LIN {X 745.357, Y -369.718, Z 305.5, A 0, B 90, C -0, E1 0, E2 0, E3 0, E4 0} C_DIS
LIN {X 743.421, Y -368.973, Z 305.5, A 0, B 90, C -0, E1 0, E2 0, E3 0, E4 0} C_DIS
LIN {X 741.486, Y -368.227, Z 305.5, A 0, B 90, C -0, E1 0, E2 0, E3 0, E4 0} C_DIS
LIN {X 739.55, Y -367.481, Z 305.5, A 0, B 90, C -0, E1 0, E2 0, E3 0, E4 0} C_DIS
LIN {X 737.563, Y -367.409, Z 305.5, A 0, B 90, C -0, E1 0, E2 0, E3 0, E4 0} C_DIS
LIN {X 736.667, Y -369.222, Z 305.5, A 0, B 90, C -0, E1 0, E2 0, E3 0, E4 0} C_DIS
LIN {X 736.176, Y -371.238, Z 305.5, A 0, B 90, C -0, E1 0, E2 0, E3 0, E4 0} C_DIS
LIN {X 735.685, Y -373.253, Z 305.5, A 0, B 90, C -0, E1 0, E2 0, E3 0, E4 0} C_DIS
LIN {X 735.194, Y -375.268, Z 305.5, A 0, B 90, C -0, E1 0, E2 0, E3 0, E4 0} C_DIS
LIN {X 734.703, Y -377.283, Z 305.5, A 0, B 90, C -0, E1 0, E2 0, E3 0, E4 0} C_DIS
LIN {X 734.212, Y -379.299, Z 305.5, A 0, B 90, C -0, E1 0, E2 0, E3 0, E4 0} C_DIS
LIN {X 733.185, Y -381.059, Z 305.5, A 0, B 90, C -0, E1 0, E2 0, E3 0, E4 0} C_DIS
LIN {X 731.276, Y -381.793, Z 305.5, A 0, B 90, C -0, E1 0, E2 0, E3 0, E4 0} C_DIS
LIN {X 729.227, Y -382.115, Z 305.5, A 0, B 90, C -0, E1 0, E2 0, E3 0, E4 0} C_DIS
LIN {X 727.178, Y -382.437, Z 305.5, A 0, B 90, C -0, E1 0, E2 0, E3 0, E4 0} C_DIS
LIN {X 725.128, Y -382.759, Z 305.5, A 0, B 90, C -0, E1 0, E2 0, E3 0, E4 0} C_DIS
LIN {X 723.079, Y -383.081, Z 305.5, A 0, B 90, C -0, E1 0, E2 0, E3 0, E4 0} C_DIS
LIN {X 721.03, Y -383.402, Z 305.5, A 0, B 90, C -0, E1 0, E2 0, E3 0, E4 0} C_DIS
LIN {X 719.273, Y -384.334, Z 305.5, A 0, B 90, C -0, E1 0, E2 0, E3 0, E4 0} C_DIS
LIN {X 719.404, Y -386.352, Z 305.5, A 0, B 90, C -0, E1 0, E2 0, E3 0, E4 0} C_DIS
LIN {X 719.987, Y -388.343, Z 305.5, A 0, B 90, C -0, E1 0, E2 0, E3 0, E4 0} C_DIS
LIN {X 720.569, Y -390.334, Z 305.5, A 0, B 90, C -0, E1 0, E2 0, E3 0, E4 0} C_DIS
LIN {X 721.151, Y -392.324, Z 305.5, A 0, B 90, C -0, E1 0, E2 0, E3 0, E4 0} C_DIS
LIN {X 721.734, Y -394.315, Z 305.5, A 0, B 90, C -0, E1 0, E2 0, E3 0, E4 0} C_DIS
LIN {X 722.316, Y -396.306, Z 305.5, A 0, B 90, C -0, E1 0, E2 0, E3 0, E4 0} C_DIS
LIN {X 722.307, Y -398.344, Z 305.5, A 0, B 90, C -0, E1 0, E2 0, E3 0, E4 0} C_DIS
LIN {X 721.021, Y -399.934, Z 305.5, A 0, B 90, C -0, E1 0, E2 0, E3 0, E4 0} C_DIS
LIN {X 719.407, Y -401.237, Z 305.5, A 0, B 90, C -0, E1 0, E2 0, E3 0, E4 0} C_DIS
LIN {X 717.793, Y -402.541, Z 305.5, A 0, B 90, C -0, E1 0, E2 0, E3 0, E4 0} C_DIS
LIN {X 716.18, Y -403.844, Z 305.5, A 0, B 90, C -0, E1 0, E2 0, E3 0, E4 0} C_DIS
LIN {X 714.566, Y -405.147, Z 305.5, A 0, B 90, C -0, E1 0, E2 0, E3 0, E4 0} C_DIS
LIN {X 712.952, Y -406.451, Z 305.5, A 0, B 90, C -0, E1 0, E2 0, E3 0, E4 0} C_DIS
LIN {X 711.897, Y -408.136, Z 305.5, A 0, B 90, C -0, E1 0, E2 0, E3 0, E4 0} C_DIS
LIN {X 713.019, Y -409.818, Z 305.5, A 0, B 90, C -0, E1 0, E2 0, E3 0, E4 0} C_DIS
LIN {X 714.519, Y -411.251, Z 305.5, A 0, B 90, C -0, E1 0, E2 0, E3 0, E4 0} C_DIS
LIN {X 716.019, Y -412.684, Z 305.5, A 0, B 90, C -0, E1 0, E2 0, E3 0, E4 0} C_DIS
LIN {X 717.518, Y -414.117, Z 305.5, A 0, B 90, C -0, E1 0, E2 0, E3 0, E4 0} C_DIS
LIN {X 719.018, Y -415.55, Z 305.5, A 0, B 90, C -0, E1 0, E2 0, E3 0, E4 0} C_DIS
LIN {X 720.518, Y -416.982, Z 305.5, A 0, B 90, C -0, E1 0, E2 0, E3 0, E4 0} C_DIS
LIN {X 721.529, Y -418.752, Z 305.5, A 0, B 90, C -0, E1 0, E2 0, E3 0, E4 0} C_DIS
LIN {X 721.21, Y -420.772, Z 305.5, A 0, B 90, C -0, E1 0, E2 0, E3 0, E4 0} C_DIS
LIN {X 720.464, Y -422.708, Z 305.5, A 0, B 90, C -0, E1 0, E2 0, E3 0, E4 0} C_DIS
LIN {X 719.718, Y -424.643, Z 305.5, A 0, B 90, C -0, E1 0, E2 0, E3 0, E4 0} C_DIS
LIN {X 718.973, Y -426.579, Z 305.5, A 0, B 90, C -0, E1 0, E2 0, E3 0, E4 0} C_DIS
LIN {X 718.227, Y -428.514, Z 305.5, A 0, B 90, C -0, E1 0, E2 0, E3 0, E4 0} C_DIS
LIN {X 717.481, Y -430.45, Z 305.5, A 0, B 90, C -0, E1 0, E2 0, E3 0, E4 0} C_DIS
LIN {X 717.409, Y -432.437, Z 305.5, A 0, B 90, C -0, E1 0, E2 0, E3 0, E4 0} C_DIS
LIN {X 719.222, Y -433.333, Z 305.5, A 0, B 90, C -0, E1 0, E2 0, E3 0, E4 0} C_DIS
LIN {X 721.238, Y -433.824, Z 305.5, A 0, B 90, C -0, E1 0, E2 0, E3 0, E4 0} C_DIS
LIN {X 723.253, Y -434.315, Z 305.5, A 0, B 90, C -0, E1 0, E2 0, E3 0, E4 0} C_DIS
LIN {X 725.268, Y -434.806, Z 305.5, A 0, B 90, C -0, E1 0, E2 0, E3 0, E4 0} C_DIS
LIN {X 727.283, Y -435.297, Z 305.5, A 0, B 90, C -0, E1 0, E2 0, E3 0, E4 0} C_DIS
LIN {X 729.299, Y -435.788, Z 305.5, A 0, B 90, C -0, E1 0, E2 0, E3 0, E4 0} C_DIS
LIN {X 731.059, Y -436.815, Z 305.5, A 0, B 90, C -0, E1 0, E2 0, E3 0, E4 0} C_DIS
LIN {X 731.793, Y -438.724, Z 305.5, A 0, B 90, C -0, E1 0, E2 0, E3 0, E4 0} C_DIS
LIN {X 732.115, Y -440.773, Z 305.5, A 0, B 90, C -0, E1 0, E2 0, E3 0, E4 0} C_DIS
LIN {X 732.437, Y -442.822, Z 305.5, A 0, B 90, C -0, E1 0, E2 0, E3 0, E4 0} C_DIS
LIN {X 732.759, Y -444.872, Z 305.5, A 0, B 90, C -0, E1 0, E2 0, E3 0, E4 0} C_DIS
LIN {X 733.081, Y -446.921, Z 305.5, A 0, B 90, C -0, E1 0, E2 0, E3 0, E4 0} C_DIS
LIN {X 733.402, Y -448.97, Z 305.5, A 0, B 90, C -0, E1 0, E2 0, E3 0, E4 0} C_DIS
LIN {X 734.334, Y -450.727, Z 305.5, A 0, B 90, C -0, E1 0, E2 0, E3 0, E4 0} C_DIS
LIN {X 736.352, Y -450.596, Z 305.5, A 0, B 90, C -0, E1 0, E2 0, E3 0, E4 0} C_DIS
LIN {X 738.343, Y -450.013, Z 305.5, A 0, B 90, C -0, E1 0, E2 0, E3 0, E4 0} C_DIS
LIN {X 740.334, Y -449.431, Z 305.5, A 0, B 90, C -0, E1 0, E2 0, E3 0, E4 0} C_DIS
LIN {X 742.324, Y -448.849, Z 305.5, A 0, B 90, C -0, E1 0, E2 0, E3 0, E4 0} C_DIS
LIN {X 744.315, Y -448.266, Z 305.5, A 0, B 90, C -0, E1 0, E2 0, E3 0, E4 0} C_DIS
LIN {X 746.306, Y -447.684, Z 305.5, A 0, B 90, C -0, E1 0, E2 0, E3 0, E4 0} C_DIS
LIN {X 748.344, Y -447.693, Z 305.5, A 0, B 90, C -0, E1 0, E2 0, E3 0, E4 0} C_DIS
LIN {X 749.934, Y -448.979, Z 305.5, A 0, B 90, C -0, E1 0, E2 0, E3 0, E4 0} C_DIS
LIN {X 751.237, Y -450.593, Z 305.5, A 0, B 90, C -0, E1 0, E2 0, E3 0, E4 0} C_DIS
LIN {X 752.541, Y -452.207, Z 305.5, A 0, B 90, C -0, E1 0, E2 0, E3 0, E4 0} C_DIS
LIN {X 753.844, Y -453.82, Z 305.5, A 0, B 90, C -0, E1 0, E2 0, E3 0, E4 0} C_DIS
LIN {X 755.147, Y -455.434, Z 305.5, A 0, B 90, C -0, E1 0, E2 0, E3 0, E4 0} C_DIS
LIN {X 756.451, Y -457.048, Z 305.5, A 0, B 90, C -0, E1 0, E2 0, E3 0, E4 0} C_DIS
LIN {X 758.136, Y -458.103, Z 305.5, A 0, B 90, C -0, E1 0, E2 0, E3 0, E4 0} C_DIS
LIN {X 759.818, Y -456.981, Z 305.5, A 0, B 90, C -0, E1 0, E2 0, E3 0, E4 0} C_DIS
LIN {X 761.251, Y -455.481, Z 305.5, A 0, B 90, C -0, E1 0, E2 0, E3 0, E4 0} C_DIS
LIN {X 762.684, Y -453.981, Z 305.5, A 0, B 90, C -0, E1 0, E2 0, E3 0, E4 0} C_DIS
LIN {X 764.117, Y -452.482, Z 305.5, A 0, B 90, C -0, E1 0, E2 0, E3 0, E4 0} C_DIS
LIN {X 765.55, Y -450.982, Z 305.5, A 0, B 90, C -0, E1 0, E2 0, E3 0, E4 0} C_DIS
LIN {X 766.982, Y -449.482, Z 305.5, A 0, B 90, C -0, E1 0, E2 0, E3 0, E4 0} C_DIS
LIN {X 768.752, Y -448.471, Z 305.5, A 0, B 90, C -0, E1 0, E2 0, E3 0, E4 0} C_DIS
LIN {X 770.772, Y -448.79, Z 305.5, A 0, B 90, C -0, E1 0, E2 0, E3 0, E4 0} C_DIS
LIN {X 772.708, Y -449.536, Z 305.5, A 0, B 90, C -0, E1 0, E2 0, E3 0, E4 0} C_DIS
LIN {X 774.643, Y -450.282, Z 305.5, A 0, B 90, C -0, E1 0, E2 0, E3 0, E4 0} C_DIS
LIN {X 776.579, Y -451.027, Z 305.5, A 0, B 90, C -0, E1 0, E2 0, E3 0, E4 0} C_DIS
LIN {X 778.514, Y -451.773, Z 305.5, A 0, B 90, C -0, E1 0, E2 0, E3 0, E4 0} C_DIS
LIN {X 780.45, Y -452.519, Z 305.5, A 0, B 90, C -0, E1 0, E2 0, E3 0, E4 0} C_DIS
LIN {X 782.437, Y -452.591, Z 305.5, A 0, B 90, C -0, E1 0, E2 0, E3 0, E4 0} C_DIS
LIN {X 783.333, Y -450.778, Z 305.5, A 0, B 90, C -0, E1 0, E2 0, E3 0, E4 0} C_DIS
LIN {X 783.824, Y -448.762, Z 305.5, A 0, B 90, C -0, E1 0, E2 0, E3 0, E4 0} C_DIS
LIN {X 784.315, Y -446.747, Z 305.5, A 0, B 90, C -0, E1 0, E2 0, E3 0, E4 0} C_DIS
LIN {X 784.806, Y -444.732, Z 305.5, A 0, B 90, C -0, E1 0, E2 0, E3 0, E4 0} C_DIS
LIN {X 785.297, Y -442.717, Z 305.5, A 0, B 90, C -0, E1 0, E2 0, E3 0, E4 0} C_DIS
LIN {X 785.788, Y -440.701, Z 305.5, A 0, B 90, C -0, E1 0, E2 0, E3 0, E4 0} C_DIS
LIN {X 786.815, Y -438.941, Z 305.5, A 0, B 90, C -0, E1 0, E2 0, E3 0, E4 0} C_DIS
LIN {X 788.724, Y -438.207, Z 305.5, A 0, B 90, C -0, E1 0, E2 0, E3 0, E4 0} C_DIS
LIN {X 790.773, Y -437.885, Z 305.5, A 0, B 90, C -0, E1 0, E2 0, E3 0, E4 0} C_DIS
LIN {X 792.822, Y -437.563, Z 305.5, A 0, B 90, C -0, E1 0, E2 0, E3 0, E4 0} C_DIS
LIN {X 794.872, Y -437.241, Z 305.5, A 0, B 90, C -0, E1 0, E2 0, E3 0, E4 0} C_DIS
LIN {X 796.921, Y -436.919, Z 305.5, A 0, B 90, C -0, E1 0, E2 0, E3 0, E4 0} C_DIS
LIN {X 798.97, Y -436.598, Z 305.5, A 0, B 90, C -0, E1 0, E2 0, E3 0, E4 0} C_DIS
LIN {X 800.727, Y -435.666, Z 305.5, A 0, B 90, C -0, E1 0, E2 0, E3 0, E4 0} C_DIS
LIN {X 800.596, Y -433.648, Z 305.5, A 0, B 90, C -0, E1 0, E2 0, E3 0, E4 0} C_DIS
LIN {X 800.013, Y -431.657, Z 305.5, A 0, B 90, C -0, E1 0, E2 0, E3 0, E4 0} C_DIS
LIN {X 799.431, Y -429.666, Z 305.5, A 0, B 90, C -0, E1 0, E2 0, E3 0, E4 0} C_DIS
LIN {X 798.849, Y -427.676, Z 305.5, A 0, B 90, C -0, E1 0, E2 0, E3 0, E4 0} C_DIS
LIN {X 798.266, Y -425.685, Z 305.5, A 0, B 90, C -0, E1 0, E2 0, E3 0, E4 0} C_DIS
LIN {X 797.684, Y -423.694, Z 305.5, A 0, B 90, C -0, E1 0, E2 0, E3 0, E4 0} C_DIS
LIN {X 797.693, Y -421.656, Z 305.5, A 0, B 90, C -0, E1 0, E2 0, E3 0, E4 0} C_DIS
LIN {X 798.979, Y -420.066, Z 305.5, A 0, B 90, C -0, E1 0, E2 0, E3 0, E4 0} C_DIS
LIN {X 800.593, Y -418.763, Z 305.5, A 0, B 90, C -0, E1 0, E2 0, E3 0, E4 0} C_DIS
LIN {X 802.207, Y -417.459, Z 305.5, A 0, B 90, C -0, E1 0, E2 0, E3 0, E4 0} C_DIS
LIN {X 803.82, Y -416.156, Z 305.5, A 0, B 90, C -0, E1 0, E2 0, E3 0, E4 0} C_DIS
LIN {X 805.434, Y -414.853, Z 305.5, A 0, B 90, C -0, E1 0, E2 0, E3 0, E4 0} C_DIS
LIN {X 807.048, Y -413.549, Z 305.5, A 0, B 90, C -0, E1 0, E2 0, E3 0, E4 0} C_DIS
LIN {X 808.103, Y -411.864, Z 305.5, A 0, B 90, C -0, E1 0, E2 0, E3 0, E4 0} C_DIS
LIN {X 806.981, Y -410.182, Z 305.5, A 0, B 90, C -0, E1 0, E2 0, E3 0, E4 0} C_DIS
LIN {X 805.481, Y -408.749, Z 305.5, A 0, B 90, C -0, E1 0, E2 0, E3 0, E4 0} C_DIS
LIN {X 803.981, Y -407.316, Z 305.5, A 0, B 90, C -0, E1 0, E2 0, E3 0, E4 0} C_DIS
LIN {X 802.482, Y -405.883, Z 305.5, A 0, B 90, C -0, E1 0, E2 0, E3 0, E4 0} C_DIS
LIN {X 800.982, Y -404.45, Z 305.5, A 0, B 90, C -0, E1 0, E2 0, E3 0, E4 0} C_DIS
LIN {X 799.482, Y -403.018, Z 305.5, A 0, B 90, C -0, E1 0, E2 0, E3 0, E4 0} C_DIS
LIN {X 798.471, Y -401.248, Z 305.5, A 0, B 90, C -0, E1 0, E2 0, E3 0, E4 0} C_DIS
LIN {X 798.79, Y -399.228, Z 305.5, A 0, B 90, C -0, E1 0, E2 0, E3 0, E4 0} C_DIS
LIN {X 799.536, Y -397.292, Z 305.5, A 0, B 90, C -0, E1 0, E2 0, E3 0, E4 0} C_DIS
LIN {X 800.282, Y -395.357, Z 305.5, A 0, B 90, C -0, E1 0, E2 0, E3 0, E4 0} C_DIS
LIN {X 801.027, Y -393.421, Z 305.5, A 0, B 90, C -0, E1 0, E2 0, E3 0, E4 0} C_DIS
LIN {X 801.773, Y -391.486, Z 305.5, A 0, B 90, C -0, E1 0, E2 0, E3 0, E4 0} C_DIS
LIN {X 802.519, Y -389.55, Z 305.5, A 0, B 90, C -0, E1 0, E2 0, E3 0, E4 0} C_DIS
LIN {X 802.591, Y -387.563, Z 305.5, A 0, B 90, C -0, E1 0, E2 0, E3 0, E4 0} C_DIS
LIN {X 800.778, Y -386.667, Z 305.5, A 0, B 90, C -0, E1 0, E2 0, E3 0, E4 0} C_DIS
LIN {X 798.762, Y -386.176, Z 305.5, A 0, B 90, C -0, E1 0, E2 0, E3 0, E4 0} C_DIS
LIN {X 796.747, Y -385.685, Z 305.5, A 0, B 90, C -0, E1 0, E2 0, E3 0, E4 0} C_DIS
LIN {X 794.732, Y -385.194, Z 305.5, A 0, B 90, C -0, E1 0, E2 0, E3 0, E4 0} C_DIS
LIN {X 792.717, Y -384.703, Z 305.5, A 0, B 90, C -0, E1 0, E2 0, E3 0, E4 0} C_DIS
LIN {X 790.701, Y -384.212, Z 305.5, A 0, B 90, C -0, E1 0, E2 0, E3 0, E4 0} C_DIS
LIN {X 788.941, Y -383.185, Z 305.5, A 0, B 90, C -0, E1 0, E2 0, E3 0, E4 0} C_DIS
LIN {X 788.207, Y -381.276, Z 305.5, A 0, B 90, C -0, E1 0, E2 0, E3 0, E4 0} C_DIS
LIN {X 787.885, Y -379.227, Z 305.5, A 0, B 90, C -0, E1 0, E2 0, E3 0, E4 0} C_DIS
LIN {X 787.563, Y -377.178, Z 305.5, A 0, B 90, C -0, E1 0, E2 0, E3 0, E4 0} C_DIS
LIN {X 787.241, Y -375.128, Z 305.5, A 0, B 90, C -0, E1 0, E2 0, E3 0, E4 0} C_DIS
LIN {X 786.919, Y -373.079, Z 305.5, A 0, B 90, C -0, E1 0, E2 0, E3 0, E4 0} C_DIS
LIN {X 786.598, Y -371.03, Z 305.5, A 0, B 90, C -0, E1 0, E2 0, E3 0, E4 0} C_DIS
LIN {X 785.666, Y -369.273, Z 305.5, A 0, B 90, C -0, E1 0, E2 0, E3 0, E4 0} C_DIS
LIN {X 783.648, Y -369.404, Z 305.5, A 0, B 90, C -0, E1 0, E2 0, E3 0, E4 0} C_DIS
LIN {X 781.657, Y -369.987, Z 305.5, A 0, B 90, C -0, E1 0, E2 0, E3 0, E4 0} C_DIS
LIN {X 779.666, Y -370.569, Z 305.5, A 0, B 90, C -0, E1 0, E2 0, E3 0, E4 0} C_DIS
LIN {X 777.676, Y -371.151, Z 305.5, A 0, B 90, C -0, E1 0, E2 0, E3 0, E4 0} C_DIS
LIN {X 775.685, Y -371.734, Z 305.5, A 0, B 90, C -0, E1 0, E2 0, E3 0, E4 0} C_DIS
LIN {X 773.694, Y -372.316, Z 305.5, A 0, B 90, C -0, E1 0, E2 0, E3 0, E4 0} C_DIS
LIN {X 771.656, Y -372.307, Z 305.5, A 0, B 90, C -0, E1 0, E2 0, E3 0, E4 0} C_DIS
LIN {X 770.066, Y -371.021, Z 305.5, A 0, B 90, C -0, E1 0, E2 0, E3 0, E4 0} C_DIS
LIN {X 768.763, Y -369.407, Z 305.5, A 0, B 90, C -0, E1 0, E2 0, E3 0, E4 0} C_DIS
LIN {X 767.459, Y -367.793, Z 305.5, A 0, B 90, C -0, E1 0, E2 0, E3 0, E4 0} C_DIS
LIN {X 766.156, Y -366.18, Z 305.5, A 0, B 90, C -0, E1 0, E2 0, E3 0, E4 0} C_DIS
LIN {X 764.853, Y -364.566, Z 305.5, A 0, B 90, C -0, E1 0, E2 0, E3 0, E4 0} C_DIS
LIN {X 763.549, Y -362.952, Z 305.5, A 0, B 90, C -0, E1 0, E2 0, E3 0, E4 0} C_DIS
LIN {X 761.864, Y -361.897, Z 305.5, A 0, B 90, C -0, E1 0, E2 0, E3 0, E4 0} C_DIS
LIN {X 760.182, Y -363.019, Z 305.5, A 0, B 90, C -0, E1 0, E2 0, E3 0, E4 0} C_DIS
LIN {X 758.749, Y -364.519, Z 305.5, A 0, B 90, C -0, E1 0, E2 0, E3 0, E4 0} C_DIS
LIN {X 757.316, Y -366.019, Z 305.5, A 0, B 90, C -0, E1 0, E2 0, E3 0, E4 0} C_DIS
LIN {X 755.883, Y -367.518, Z 305.5, A 0, B 90, C -0, E1 0, E2 0, E3 0, E4 0} C_DIS
LIN {X 754.45, Y -369.018, Z 305.5, A 0, B 90, C -0, E1 0, E2 0, E3 0, E4 0} C_DIS
LIN {X 752.899, Y -370.544, Z 306.8, A 0, B 90, C -0, E1 0, E2 0, E3 0, E4 0} C_DIS
LIN {X 751.133, Y -371.56, Z 306.8, A 0, B 90, C -0, E1 0, E2 0, E3 0, E4 0} C_DIS
LIN {X 749.112, Y -371.247, Z 306.8, A 0, B 90, C -0, E1 0, E2 0, E3 0, E4 0} C_DIS
LIN {X 747.174, Y -370.508, Z 306.8, A 0, B 90, C -0, E1 0, E2 0, E3 0, E4 0} C_DIS
LIN {X 745.237, Y -369.768, Z 306.8, A 0, B 90, C -0, E1 0, E2 0, E3 0, E4 0} C_DIS
LIN {X 743.299, Y -369.028, Z 306.8, A 0, B 90, C -0, E1 0, E2 0, E3 0, E4 0} C_DIS
LIN {X 741.362, Y -368.288, Z 306.8, A 0, B 90, C -0, E1 0, E2 0, E3 0, E4 0} C_DIS
LIN {X 739.424, Y -367.548, Z 306.8, A 0, B 90, C -0, E1 0, E2 0, E3 0, E4 0} C_DIS
LIN {X 737.437, Y -367.482, Z 306.8, A 0, B 90, C -0, E1 0, E2 0, E3 0, E4 0} C_DIS
LIN {X 736.547, Y -369.298, Z 306.8, A 0, B 90, C -0, E1 0, E2 0, E3 0, E4 0} C_DIS
LIN {X 736.062, Y -371.315, Z 306.8, A 0, B 90, C -0, E1 0, E2 0, E3 0, E4 0} C_DIS
LIN {X 735.577, Y -373.331, Z 306.8, A 0, B 90, C -0, E1 0, E2 0, E3 0, E4 0} C_DIS
LIN {X 735.092, Y -375.348, Z 306.8, A 0, B 90, C -0, E1 0, E2 0, E3 0, E4 0} C_DIS
LIN {X 734.607, Y -377.364, Z 306.8, A 0, B 90, C -0, E1 0, E2 0, E3 0, E4 0} C_DIS
LIN {X 734.123, Y -379.381, Z 306.8, A 0, B 90, C -0, E1 0, E2 0, E3 0, E4 0} C_DIS
LIN {X 733.101, Y -381.144, Z 306.8, A 0, B 90, C -0, E1 0, E2 0, E3 0, E4 0} C_DIS
LIN {X 731.194, Y -381.883, Z 306.8, A 0, B 90, C -0, E1 0, E2 0, E3 0, E4 0} C_DIS
LIN {X 729.147, Y -382.211, Z 306.8, A 0, B 90, C -0, E1 0, E2 0, E3 0, E4 0} C_DIS
LIN {X 727.099, Y -382.539, Z 306.8, A 0, B 90, C -0, E1 0, E2 0, E3 0, E4 0} C_DIS
LIN {X 725.051, Y -382.867, Z 306.8, A 0, B 90, C -0, E1 0, E2 0, E3 0, E4 0} C_DIS
LIN {X 723.003, Y -383.195, Z 306.8, A 0, B 90, C -0, E1 0, E2 0, E3 0, E4 0} C_DIS
LIN {X 720.955, Y -383.523, Z 306.8, A 0, B 90, C -0, E1 0, E2 0, E3 0, E4 0} C_DIS
LIN {X 719.201, Y -384.46, Z 306.8, A 0, B 90, C -0, E1 0, E2 0, E3 0, E4 0} C_DIS
LIN {X 719.338, Y -386.478, Z 306.8, A 0, B 90, C -0, E1 0, E2 0, E3 0, E4 0} C_DIS
LIN {X 719.926, Y -388.466, Z 306.8, A 0, B 90, C -0, E1 0, E2 0, E3 0, E4 0} C_DIS
LIN {X 720.515, Y -390.455, Z 306.8, A 0, B 90, C -0, E1 0, E2 0, E3 0, E4 0} C_DIS
LIN {X 721.103, Y -392.444, Z 306.8, A 0, B 90, C -0, E1 0, E2 0, E3 0, E4 0} C_DIS
LIN {X 721.691, Y -394.433, Z 306.8, A 0, B 90, C -0, E1 0, E2 0, E3 0, E4 0} C_DIS
LIN {X 722.28, Y -396.421, Z 306.8, A 0, B 90, C -0, E1 0, E2 0, E3 0, E4 0} C_DIS
LIN {X 722.277, Y -398.459, Z 306.8, A 0, B 90, C -0, E1 0, E2 0, E3 0, E4 0} C_DIS
LIN {X 720.995, Y -400.053, Z 306.8, A 0, B 90, C -0, E1 0, E2 0, E3 0, E4 0} C_DIS
LIN {X 719.386, Y -401.361, Z 306.8, A 0, B 90, C -0, E1 0, E2 0, E3 0, E4 0} C_DIS
LIN {X 717.776, Y -402.669, Z 306.8, A 0, B 90, C -0, E1 0, E2 0, E3 0, E4 0} C_DIS
LIN {X 716.167, Y -403.977, Z 306.8, A 0, B 90, C -0, E1 0, E2 0, E3 0, E4 0} C_DIS
LIN {X 714.557, Y -405.285, Z 306.8, A 0, B 90, C -0, E1 0, E2 0, E3 0, E4 0} C_DIS
LIN {X 712.948, Y -406.593, Z 306.8, A 0, B 90, C -0, E1 0, E2 0, E3 0, E4 0} C_DIS
LIN {X 711.897, Y -408.281, Z 306.8, A 0, B 90, C -0, E1 0, E2 0, E3 0, E4 0} C_DIS
LIN {X 713.025, Y -409.96, Z 306.8, A 0, B 90, C -0, E1 0, E2 0, E3 0, E4 0} C_DIS
LIN {X 714.529, Y -411.388, Z 306.8, A 0, B 90, C -0, E1 0, E2 0, E3 0, E4 0} C_DIS
LIN {X 716.032, Y -412.816, Z 306.8, A 0, B 90, C -0, E1 0, E2 0, E3 0, E4 0} C_DIS
LIN {X 717.536, Y -414.244, Z 306.8, A 0, B 90, C -0, E1 0, E2 0, E3 0, E4 0} C_DIS
LIN {X 719.04, Y -415.673, Z 306.8, A 0, B 90, C -0, E1 0, E2 0, E3 0, E4 0} C_DIS
LIN {X 720.544, Y -417.101, Z 306.8, A 0, B 90, C -0, E1 0, E2 0, E3 0, E4 0} C_DIS
LIN {X 721.56, Y -418.867, Z 306.8, A 0, B 90, C -0, E1 0, E2 0, E3 0, E4 0} C_DIS
LIN {X 721.247, Y -420.888, Z 306.8, A 0, B 90, C -0, E1 0, E2 0, E3 0, E4 0} C_DIS
LIN {X 720.508, Y -422.826, Z 306.8, A 0, B 90, C -0, E1 0, E2 0, E3 0, E4 0} C_DIS
LIN {X 719.768, Y -424.763, Z 306.8, A 0, B 90, C -0, E1 0, E2 0, E3 0, E4 0} C_DIS
LIN {X 719.028, Y -426.701, Z 306.8, A 0, B 90, C -0, E1 0, E2 0, E3 0, E4 0} C_DIS
LIN {X 718.288, Y -428.638, Z 306.8, A 0, B 90, C -0, E1 0, E2 0, E3 0, E4 0} C_DIS
LIN {X 717.548, Y -430.576, Z 306.8, A 0, B 90, C -0, E1 0, E2 0, E3 0, E4 0} C_DIS
LIN {X 717.482, Y -432.563, Z 306.8, A 0, B 90, C -0, E1 0, E2 0, E3 0, E4 0} C_DIS
LIN {X 719.298, Y -433.453, Z 306.8, A 0, B 90, C -0, E1 0, E2 0, E3 0, E4 0} C_DIS
LIN {X 721.315, Y -433.938, Z 306.8, A 0, B 90, C -0, E1 0, E2 0, E3 0, E4 0} C_DIS
LIN {X 723.331, Y -434.423, Z 306.8, A 0, B 90, C -0, E1 0, E2 0, E3 0, E4 0} C_DIS
LIN {X 725.348, Y -434.908, Z 306.8, A 0, B 90, C -0, E1 0, E2 0, E3 0, E4 0} C_DIS
LIN {X 727.364, Y -435.392, Z 306.8, A 0, B 90, C -0, E1 0, E2 0, E3 0, E4 0} C_DIS
LIN {X 729.381, Y -435.877, Z 306.8, A 0, B 90, C -0, E1 0, E2 0, E3 0, E4 0} C_DIS
LIN {X 731.144, Y -436.899, Z 306.8, A 0, B 90, C -0, E1 0, E2 0, E3 0, E4 0} C_DIS
LIN {X 731.883, Y -438.806, Z 306.8, A 0, B 90, C -0, E1 0, E2 0, E3 0, E4 0} C_DIS
LIN {X 732.211, Y -440.853, Z 306.8, A 0, B 90, C -0, E1 0, E2 0, E3 0, E4 0} C_DIS
LIN {X 732.539, Y -442.901, Z 306.8, A 0, B 90, C -0, E1 0, E2 0, E3 0, E4 0} C_DIS
LIN {X 732.867, Y -444.949, Z 306.8, A 0, B 90, C -0, E1 0, E2 0, E3 0, E4 0} C_DIS
LIN {X 733.195, Y -446.997, Z 306.8, A 0, B 90, C -0, E1 0, E2 0, E3 0, E4 0} C_DIS
LIN {X 733.523, Y -449.045, Z 306.8, A 0, B 90, C -0, E1 0, E2 0, E3 0, E4 0} C_DIS
LIN {X 734.46, Y -450.799, Z 306.8, A 0, B 90, C -0, E1 0, E2 0, E3 0, E4 0} C_DIS
LIN {X 736.478, Y -450.662, Z 306.8, A 0, B 90, C -0, E1 0, E2 0, E3 0, E4 0} C_DIS
LIN {X 738.466, Y -450.074, Z 306.8, A 0, B 90, C -0, E1 0, E2 0, E3 0, E4 0} C_DIS
LIN {X 740.455, Y -449.485, Z 306.8, A 0, B 90, C -0, E1 0, E2 0, E3 0, E4 0} C_DIS
LIN {X 742.444, Y -448.897, Z 306.8, A 0, B 90, C -0, E1 0, E2 0, E3 0, E4 0} C_DIS
LIN {X 744.433, Y -448.309, Z 306.8, A 0, B 90, C -0, E1 0, E2 0, E3 0, E4 0} C_DIS
LIN {X 746.421, Y -447.72, Z 306.8, A 0, B 90, C -0, E1 0, E2 0, E3 0, E4 0} C_DIS
LIN {X 748.459, Y -447.723, Z 306.8, A 0, B 90, C -0, E1 0, E2 0, E3 0, E4 0} C_DIS
LIN {X 750.053, Y -449.005, Z 306.8, A 0, B 90, C -0, E1 0, E2 0, E3 0, E4 0} C_DIS
LIN {X 751.361, Y -450.614, Z 306.8, A 0, B 90, C -0, E1 0, E2 0, E3 0, E4 0} C_DIS
LIN {X 752.669, Y -452.224, Z 306.8, A 0, B 90, C -0, E1 0, E2 0, E3 0, E4 0} C_DIS
LIN {X 753.977, Y -453.833, Z 306.8, A 0, B 90, C -0, E1 0, E2 0, E3 0, E4 0} C_DIS
LIN {X 755.285, Y -455.443, Z 306.8, A 0, B 90, C -0, E1 0, E2 0, E3 0, E4 0} C_DIS
LIN {X 756.593, Y -457.052, Z 306.8, A 0, B 90, C -0, E1 0, E2 0, E3 0, E4 0} C_DIS
LIN {X 758.281, Y -458.103, Z 306.8, A 0, B 90, C -0, E1 0, E2 0, E3 0, E4 0} C_DIS
LIN {X 759.96, Y -456.975, Z 306.8, A 0, B 90, C -0, E1 0, E2 0, E3 0, E4 0} C_DIS
LIN {X 761.388, Y -455.471, Z 306.8, A 0, B 90, C -0, E1 0, E2 0, E3 0, E4 0} C_DIS
LIN {X 762.816, Y -453.968, Z 306.8, A 0, B 90, C -0, E1 0, E2 0, E3 0, E4 0} C_DIS
LIN {X 764.244, Y -452.464, Z 306.8, A 0, B 90, C -0, E1 0, E2 0, E3 0, E4 0} C_DIS
LIN {X 765.673, Y -450.96, Z 306.8, A 0, B 90, C -0, E1 0, E2 0, E3 0, E4 0} C_DIS
LIN {X 767.101, Y -449.456, Z 306.8, A 0, B 90, C -0, E1 0, E2 0, E3 0, E4 0} C_DIS
LIN {X 768.867, Y -448.44, Z 306.8, A 0, B 90, C -0, E1 0, E2 0, E3 0, E4 0} C_DIS
LIN {X 770.888, Y -448.753, Z 306.8, A 0, B 90, C -0, E1 0, E2 0, E3 0, E4 0} C_DIS
LIN {X 772.826, Y -449.492, Z 306.8, A 0, B 90, C -0, E1 0, E2 0, E3 0, E4 0} C_DIS
LIN {X 774.763, Y -450.232, Z 306.8, A 0, B 90, C -0, E1 0, E2 0, E3 0, E4 0} C_DIS
LIN {X 776.701, Y -450.972, Z 306.8, A 0, B 90, C -0, E1 0, E2 0, E3 0, E4 0} C_DIS
LIN {X 778.638, Y -451.712, Z 306.8, A 0, B 90, C -0, E1 0, E2 0, E3 0, E4 0} C_DIS
LIN {X 780.576, Y -452.452, Z 306.8, A 0, B 90, C -0, E1 0, E2 0, E3 0, E4 0} C_DIS
LIN {X 782.563, Y -452.518, Z 306.8, A 0, B 90, C -0, E1 0, E2 0, E3 0, E4 0} C_DIS
LIN {X 783.453, Y -450.702, Z 306.8, A 0, B 90, C -0, E1 0, E2 0, E3 0, E4 0} C_DIS
LIN {X 783.938, Y -448.685, Z 306.8, A 0, B 90, C -0, E1 0, E2 0, E3 0, E4 0} C_DIS
LIN {X 784.423, Y -446.669, Z 306.8, A 0, B 90, C -0, E1 0, E2 0, E3 0, E4 0} C_DIS
LIN {X 784.908, Y -444.652, Z 306.8, A 0, B 90, C -0, E1 0, E2 0, E3 0, E4 0} C_DIS
LIN {X 785.393, Y -442.636, Z 306.8, A 0, B 90, C -0, E1 0, E2 0, E3 0, E4 0} C_DIS
LIN {X 785.877, Y -440.619, Z 306.8, A 0, B 90, C -0, E1 0, E2 0, E3 0, E4 0} C_DIS
LIN {X 786.899, Y -438.856, Z 306.8, A 0, B 90, C -0, E1 0, E2 0, E3 0, E4 0} C_DIS
LIN {X 788.806, Y -438.117, Z 306.8, A 0, B 90, C -0, E1 0, E2 0, E3 0, E4 0} C_DIS
LIN {X 790.853, Y -437.789, Z 306.8, A 0, B 90, C -0, E1 0, E2 0, E3 0, E4 0} C_DIS
LIN {X 792.901, Y -437.461, Z 306.8, A 0, B 90, C -0, E1 0, E2 0, E3 0, E4 0} C_DIS
LIN {X 794.949, Y -437.133, Z 306.8, A 0, B 90, C -0, E1 0, E2 0, E3 0, E4 0} C_DIS
LIN {X 796.997, Y -436.805, Z 306.8, A 0, B 90, C -0, E1 0, E2 0, E3 0, E4 0} C_DIS
LIN {X 799.045, Y -436.477, Z 306.8, A 0, B 90, C -0, E1 0, E2 0, E3 0, E4 0} C_DIS
LIN {X 800.799, Y -435.54, Z 306.8, A 0, B 90, C -0, E1 0, E2 0, E3 0, E4 0} C_DIS
LIN {X 800.662, Y -433.522, Z 306.8, A 0, B 90, C -0, E1 0, E2 0, E3 0, E4 0} C_DIS
LIN {X 800.074, Y -431.534, Z 306.8, A 0, B 90, C -0, E1 0, E2 0, E3 0, E4 0} C_DIS
LIN {X 799.485, Y -429.545, Z 306.8, A 0, B 90, C -0, E1 0, E2 0, E3 0, E4 0} C_DIS
LIN {X 798.897, Y -427.556, Z 306.8, A 0, B 90, C -0, E1 0, E2 0, E3 0, E4 0} C_DIS
LIN {X 798.309, Y -425.567, Z 306.8, A 0, B 90, C -0, E1 0, E2 0, E3 0, E4 0} C_DIS
LIN {X 797.72, Y -423.579, Z 306.8, A 0, B 90, C -0, E1 0, E2 0, E3 0, E4 0} C_DIS
LIN {X 797.723, Y -421.541, Z 306.8, A 0, B 90, C -0, E1 0, E2 0, E3 0, E4 0} C_DIS
LIN {X 799.005, Y -419.947, Z 306.8, A 0, B 90, C -0, E1 0, E2 0, E3 0, E4 0} C_DIS
LIN {X 800.614, Y -418.639, Z 306.8, A 0, B 90, C -0, E1 0, E2 0, E3 0, E4 0} C_DIS
LIN {X 802.224, Y -417.331, Z 306.8, A 0, B 90, C -0, E1 0, E2 0, E3 0, E4 0} C_DIS
LIN {X 803.833, Y -416.023, Z 306.8, A 0, B 90, C -0, E1 0, E2 0, E3 0, E4 0} C_DIS
LIN {X 805.443, Y -414.715, Z 306.8, A 0, B 90, C -0, E1 0, E2 0, E3 0, E4 0} C_DIS
LIN {X 807.052, Y -413.407, Z 306.8, A 0, B 90, C -0, E1 0, E2 0, E3 0, E4 0} C_DIS
LIN {X 808.103, Y -411.719, Z 306.8, A 0, B 90, C -0, E1 0, E2 0, E3 0, E4 0} C_DIS
LIN {X 806.975, Y -410.04, Z 306.8, A 0, B 90, C -0, E1 0, E2 0, E3 0, E4 0} C_DIS
LIN {X 805.471, Y -408.612, Z 306.8, A 0, B 90, C -0, E1 0, E2 0, E3 0, E4 0} C_DIS
LIN {X 803.968, Y -407.184, Z 306.8, A 0, B 90, C -0, E1 0, E2 0, E3 0, E4 0} C_DIS
LIN {X 802.464, Y -405.756, Z 306.8, A 0, B 90, C -0, E1 0, E2 0, E3 0, E4 0} C_DIS
LIN {X 800.96, Y -404.327, Z 306.8, A 0, B 90, C -0, E1 0, E2 0, E3 0, E4 0} C_DIS
LIN {X 799.456, Y -402.899, Z 306.8, A 0, B 90, C -0, E1 0, E2 0, E3 0, E4 0} C_DIS
LIN {X 798.44, Y -401.133, Z 306.8, A 0, B 90, C -0, E1 0, E2 0, E3 0, E4 0} C_DIS
LIN {X 798.753, Y -399.112, Z 306.8, A 0, B 90, C -0, E1 0, E2 0, E3 0, E4 0} C_DIS
LIN {X 799.492, Y -397.174, Z 306.8, A 0, B 90, C -0, E1 0, E2 0, E3 0, E4 0} C_DIS
LIN {X 800.232, Y -395.237, Z 306.8, A 0, B 90, C -0, E1 0, E2 0, E3 0, E4 0} C_DIS
LIN {X 800.972, Y -393.299, Z 306.8, A 0, B 90, C -0, E1 0, E2 0, E3 0, E4 0} C_DIS
LIN {X 801.712, Y -391.362, Z 306.8, A 0, B 90, C -0, E1 0, E2 0, E3 0, E4 0} C_DIS
LIN {X 802.452, Y -389.424, Z 306.8, A 0, B 90, C -0, E1 0, E2 0, E3 0, E4 0} C_DIS
LIN {X 802.518, Y -387.437, Z 306.8, A 0, B 90, C -0, E1 0, E2 0, E3 0, E4 0} C_DIS
LIN {X 800.702, Y -386.547, Z 306.8, A 0, B 90, C -0, E1 0, E2 0, E3 0, E4 0} C_DIS
LIN {X 798.685, Y -386.062, Z 306.8, A 0, B 90, C -0, E1 0, E2 0, E3 0, E4 0} C_DIS
LIN {X 796.669, Y -385.577, Z 306.8, A 0, B 90, C -0, E1 0, E2 0, E3 0, E4 0} C_DIS
LIN {X 794.652, Y -385.092, Z 306.8, A 0, B 90, C -0, E1 0, E2 0, E3 0, E4 0} C_DIS
LIN {X 792.636, Y -384.608, Z 306.8, A 0, B 90, C -0, E1 0, E2 0, E3 0, E4 0} C_DIS
LIN {X 790.619, Y -384.123, Z 306.8, A 0, B 90, C -0, E1 0, E2 0, E3 0, E4 0} C_DIS
LIN {X 788.856, Y -383.101, Z 306.8, A 0, B 90, C -0, E1 0, E2 0, E3 0, E4 0} C_DIS
LIN {X 788.117, Y -381.194, Z 306.8, A 0, B 90, C -0, E1 0, E2 0, E3 0, E4 0} C_DIS
LIN {X 787.789, Y -379.147, Z 306.8, A 0, B 90, C -0, E1 0, E2 0, E3 0, E4 0} C_DIS
LIN {X 787.461, Y -377.099, Z 306.8, A 0, B 90, C -0, E1 0, E2 0, E3 0, E4 0} C_DIS
LIN {X 787.133, Y -375.051, Z 306.8, A 0, B 90, C -0, E1 0, E2 0, E3 0, E4 0} C_DIS
LIN {X 786.805, Y -373.003, Z 306.8, A 0, B 90, C -0, E1 0, E2 0, E3 0, E4 0} C_DIS
LIN {X 786.477, Y -370.955, Z 306.8, A 0, B 90, C -0, E1 0, E2 0, E3 0, E4 0} C_DIS
LIN {X 785.54, Y -369.201, Z 306.8, A 0, B 90, C -0, E1 0, E2 0, E3 0, E4 0} C_DIS
LIN {X 783.522, Y -369.338, Z 306.8, A 0, B 90, C -0, E1 0, E2 0, E3 0, E4 0} C_DIS
LIN {X 781.534, Y -369.926, Z 306.8, A 0, B 90, C -0, E1 0, E2 0, E3 0, E4 0} C_DIS
LIN {X 779.545, Y -370.515, Z 306.8, A 0, B 90, C -0, E1 0, E2 0, E3 0, E4 0} C_DIS
LIN {X 777.556, Y -371.103, Z 306.8, A 0, B 90, C -0, E1 0, E2 0, E3 0, E4 0} C_DIS
LIN {X 775.567, Y -371.691, Z 306.8, A 0, B 90, C -0, E1 0, E2 0, E3 0, E4 0} C_DIS
LIN {X 773.579, Y -372.28, Z 306.8, A 0, B 90, C -0, E1 0, E2 0, E3 0, E4 0} C_DIS
LIN {X 771.541, Y -372.277, Z 306.8, A 0, B 90, C -0, E1 0, E2 0, E3 0, E4 0} C_DIS
LIN {X 769.947, Y -370.995, Z 306.8, A 0, B 90, C -0, E1 0, E2 0, E3 0, E4 0} C_DIS
LIN {X 768.639, Y -369.386, Z 306.8, A 0, B 90, C -0, E1 0, E2 0, E3 0, E4 0} C_DIS
LIN {X 767.331, Y -367.776, Z 306.8, A 0, B 90, C -0, E1 0, E2 0, E3 0, E4 0} C_DIS
LIN {X 766.023, Y -366.167, Z 306.8, A 0, B 90, C -0, E1 0, E2 0, E3 0, E4 0} C_DIS
LIN {X 764.715, Y -364.557, Z 306.8, A 0, B 90, C -0, E1 0, E2 0, E3 0, E4 0} C_DIS
LIN {X 763.407, Y -362.948, Z 306.8, A 0, B 90, C -0, E1 0, E2 0, E3 0, E4 0} C_DIS
LIN {X 761.719, Y -361.897, Z 306.8, A 0, B 90, C -0, E1 0, E2 0, E3 0, E4 0} C_DIS
LIN {X 760.04, Y -363.025, Z 306.8, A 0, B 90, C -0, E1 0, E2 0, E3 0, E4 0} C_DIS
LIN {X 758.612, Y -364.529, Z 306.8, A 0, B 90, C -0, E1 0, E2 0, E3 0, E4 0} C_DIS
LIN {X 757.184, Y -366.032, Z 306.8, A 0, B 90, C -0, E1 0, E2 0, E3 0, E4 0} C_DIS
LIN {X 755.756, Y -367.536, Z 306.8, A 0, B 90, C -0, E1 0, E2 0, E3 0, E4 0} C_DIS
LIN {X 754.327, Y -369.04, Z 306.8, A 0, B 90, C -0, E1 0, E2 0, E3 0, E4 0} C_DIS
LIN {X 752.785, Y -370.567, Z 308.1, A 0, B 90, C -0, E1 0, E2 0, E3 0, E4 0} C_DIS
LIN {X 751.021, Y -371.588, Z 308.1, A 0, B 90, C -0, E1 0, E2 0, E3 0, E4 0} C_DIS
LIN {X 749, Y -371.281, Z 308.1, A 0, B 90, C -0, E1 0, E2 0, E3 0, E4 0} C_DIS
LIN {X 747.06, Y -370.547, Z 308.1, A 0, B 90, C -0, E1 0, E2 0, E3 0, E4 0} C_DIS
LIN {X 745.121, Y -369.813, Z 308.1, A 0, B 90, C -0, E1 0, E2 0, E3 0, E4 0} C_DIS
LIN {X 743.181, Y -369.079, Z 308.1, A 0, B 90, C -0, E1 0, E2 0, E3 0, E4 0} C_DIS
LIN {X 741.242, Y -368.345, Z 308.1, A 0, B 90, C -0, E1 0, E2 0, E3 0, E4 0} C_DIS
LIN {X 739.302, Y -367.611, Z 308.1, A 0, B 90, C -0, E1 0, E2 0, E3 0, E4 0} C_DIS
LIN {X 737.315, Y -367.55, Z 308.1, A 0, B 90, C -0, E1 0, E2 0, E3 0, E4 0} C_DIS
LIN {X 736.43, Y -369.369, Z 308.1, A 0, B 90, C -0, E1 0, E2 0, E3 0, E4 0} C_DIS
LIN {X 735.951, Y -371.387, Z 308.1, A 0, B 90, C -0, E1 0, E2 0, E3 0, E4 0} C_DIS
LIN {X 735.472, Y -373.404, Z 308.1, A 0, B 90, C -0, E1 0, E2 0, E3 0, E4 0} C_DIS
LIN {X 734.993, Y -375.422, Z 308.1, A 0, B 90, C -0, E1 0, E2 0, E3 0, E4 0} C_DIS
LIN {X 734.514, Y -377.44, Z 308.1, A 0, B 90, C -0, E1 0, E2 0, E3 0, E4 0} C_DIS
LIN {X 734.035, Y -379.458, Z 308.1, A 0, B 90, C -0, E1 0, E2 0, E3 0, E4 0} C_DIS
LIN {X 733.018, Y -381.224, Z 308.1, A 0, B 90, C -0, E1 0, E2 0, E3 0, E4 0} C_DIS
LIN {X 731.114, Y -381.969, Z 308.1, A 0, B 90, C -0, E1 0, E2 0, E3 0, E4 0} C_DIS
LIN {X 729.067, Y -382.303, Z 308.1, A 0, B 90, C -0, E1 0, E2 0, E3 0, E4 0} C_DIS
LIN {X 727.021, Y -382.637, Z 308.1, A 0, B 90, C -0, E1 0, E2 0, E3 0, E4 0} C_DIS
LIN {X 724.974, Y -382.971, Z 308.1, A 0, B 90, C -0, E1 0, E2 0, E3 0, E4 0} C_DIS
LIN {X 722.927, Y -383.305, Z 308.1, A 0, B 90, C -0, E1 0, E2 0, E3 0, E4 0} C_DIS
LIN {X 720.88, Y -383.639, Z 308.1, A 0, B 90, C -0, E1 0, E2 0, E3 0, E4 0} C_DIS
LIN {X 719.129, Y -384.58, Z 308.1, A 0, B 90, C -0, E1 0, E2 0, E3 0, E4 0} C_DIS
LIN {X 719.272, Y -386.597, Z 308.1, A 0, B 90, C -0, E1 0, E2 0, E3 0, E4 0} C_DIS
LIN {X 719.866, Y -388.584, Z 308.1, A 0, B 90, C -0, E1 0, E2 0, E3 0, E4 0} C_DIS
LIN {X 720.46, Y -390.571, Z 308.1, A 0, B 90, C -0, E1 0, E2 0, E3 0, E4 0} C_DIS
LIN {X 721.054, Y -392.558, Z 308.1, A 0, B 90, C -0, E1 0, E2 0, E3 0, E4 0} C_DIS
LIN {X 721.648, Y -394.545, Z 308.1, A 0, B 90, C -0, E1 0, E2 0, E3 0, E4 0} C_DIS
LIN {X 722.242, Y -396.532, Z 308.1, A 0, B 90, C -0, E1 0, E2 0, E3 0, E4 0} C_DIS
LIN {X 722.245, Y -398.57, Z 308.1, A 0, B 90, C -0, E1 0, E2 0, E3 0, E4 0} C_DIS
LIN {X 720.969, Y -400.167, Z 308.1, A 0, B 90, C -0, E1 0, E2 0, E3 0, E4 0} C_DIS
LIN {X 719.363, Y -401.48, Z 308.1, A 0, B 90, C -0, E1 0, E2 0, E3 0, E4 0} C_DIS
LIN {X 717.757, Y -402.792, Z 308.1, A 0, B 90, C -0, E1 0, E2 0, E3 0, E4 0} C_DIS
LIN {X 716.152, Y -404.105, Z 308.1, A 0, B 90, C -0, E1 0, E2 0, E3 0, E4 0} C_DIS
LIN {X 714.546, Y -405.418, Z 308.1, A 0, B 90, C -0, E1 0, E2 0, E3 0, E4 0} C_DIS
LIN {X 712.941, Y -406.73, Z 308.1, A 0, B 90, C -0, E1 0, E2 0, E3 0, E4 0} C_DIS
LIN {X 711.895, Y -408.421, Z 308.1, A 0, B 90, C -0, E1 0, E2 0, E3 0, E4 0} C_DIS
LIN {X 713.027, Y -410.097, Z 308.1, A 0, B 90, C -0, E1 0, E2 0, E3 0, E4 0} C_DIS
LIN {X 714.535, Y -411.52, Z 308.1, A 0, B 90, C -0, E1 0, E2 0, E3 0, E4 0} C_DIS
LIN {X 716.043, Y -412.944, Z 308.1, A 0, B 90, C -0, E1 0, E2 0, E3 0, E4 0} C_DIS
LIN {X 717.551, Y -414.368, Z 308.1, A 0, B 90, C -0, E1 0, E2 0, E3 0, E4 0} C_DIS
LIN {X 719.059, Y -415.792, Z 308.1, A 0, B 90, C -0, E1 0, E2 0, E3 0, E4 0} C_DIS
LIN {X 720.567, Y -417.215, Z 308.1, A 0, B 90, C -0, E1 0, E2 0, E3 0, E4 0} C_DIS
LIN {X 721.588, Y -418.979, Z 308.1, A 0, B 90, C -0, E1 0, E2 0, E3 0, E4 0} C_DIS
LIN {X 721.281, Y -421, Z 308.1, A 0, B 90, C -0, E1 0, E2 0, E3 0, E4 0} C_DIS
LIN {X 720.547, Y -422.94, Z 308.1, A 0, B 90, C -0, E1 0, E2 0, E3 0, E4 0} C_DIS
LIN {X 719.813, Y -424.879, Z 308.1, A 0, B 90, C -0, E1 0, E2 0, E3 0, E4 0} C_DIS
LIN {X 719.079, Y -426.819, Z 308.1, A 0, B 90, C -0, E1 0, E2 0, E3 0, E4 0} C_DIS
LIN {X 718.345, Y -428.758, Z 308.1, A 0, B 90, C -0, E1 0, E2 0, E3 0, E4 0} C_DIS
LIN {X 717.611, Y -430.698, Z 308.1, A 0, B 90, C -0, E1 0, E2 0, E3 0, E4 0} C_DIS
LIN {X 717.55, Y -432.685, Z 308.1, A 0, B 90, C -0, E1 0, E2 0, E3 0, E4 0} C_DIS
LIN {X 719.369, Y -433.57, Z 308.1, A 0, B 90, C -0, E1 0, E2 0, E3 0, E4 0} C_DIS
LIN {X 721.387, Y -434.049, Z 308.1, A 0, B 90, C -0, E1 0, E2 0, E3 0, E4 0} C_DIS
LIN {X 723.404, Y -434.528, Z 308.1, A 0, B 90, C -0, E1 0, E2 0, E3 0, E4 0} C_DIS
LIN {X 725.422, Y -435.007, Z 308.1, A 0, B 90, C -0, E1 0, E2 0, E3 0, E4 0} C_DIS
LIN {X 727.44, Y -435.486, Z 308.1, A 0, B 90, C -0, E1 0, E2 0, E3 0, E4 0} C_DIS
LIN {X 729.458, Y -435.965, Z 308.1, A 0, B 90, C -0, E1 0, E2 0, E3 0, E4 0} C_DIS
LIN {X 731.224, Y -436.982, Z 308.1, A 0, B 90, C -0, E1 0, E2 0, E3 0, E4 0} C_DIS
LIN {X 731.969, Y -438.886, Z 308.1, A 0, B 90, C -0, E1 0, E2 0, E3 0, E4 0} C_DIS
LIN {X 732.303, Y -440.933, Z 308.1, A 0, B 90, C -0, E1 0, E2 0, E3 0, E4 0} C_DIS
LIN {X 732.637, Y -442.979, Z 308.1, A 0, B 90, C -0, E1 0, E2 0, E3 0, E4 0} C_DIS
LIN {X 732.971, Y -445.026, Z 308.1, A 0, B 90, C -0, E1 0, E2 0, E3 0, E4 0} C_DIS
LIN {X 733.305, Y -447.073, Z 308.1, A 0, B 90, C -0, E1 0, E2 0, E3 0, E4 0} C_DIS
LIN {X 733.639, Y -449.12, Z 308.1, A 0, B 90, C -0, E1 0, E2 0, E3 0, E4 0} C_DIS
LIN {X 734.58, Y -450.871, Z 308.1, A 0, B 90, C -0, E1 0, E2 0, E3 0, E4 0} C_DIS
LIN {X 736.597, Y -450.728, Z 308.1, A 0, B 90, C -0, E1 0, E2 0, E3 0, E4 0} C_DIS
LIN {X 738.584, Y -450.134, Z 308.1, A 0, B 90, C -0, E1 0, E2 0, E3 0, E4 0} C_DIS
LIN {X 740.571, Y -449.54, Z 308.1, A 0, B 90, C -0, E1 0, E2 0, E3 0, E4 0} C_DIS
LIN {X 742.558, Y -448.946, Z 308.1, A 0, B 90, C -0, E1 0, E2 0, E3 0, E4 0} C_DIS
LIN {X 744.545, Y -448.352, Z 308.1, A 0, B 90, C -0, E1 0, E2 0, E3 0, E4 0} C_DIS
LIN {X 746.532, Y -447.758, Z 308.1, A 0, B 90, C -0, E1 0, E2 0, E3 0, E4 0} C_DIS
LIN {X 748.57, Y -447.755, Z 308.1, A 0, B 90, C -0, E1 0, E2 0, E3 0, E4 0} C_DIS
LIN {X 750.167, Y -449.031, Z 308.1, A 0, B 90, C -0, E1 0, E2 0, E3 0, E4 0} C_DIS
LIN {X 751.48, Y -450.637, Z 308.1, A 0, B 90, C -0, E1 0, E2 0, E3 0, E4 0} C_DIS
LIN {X 752.792, Y -452.243, Z 308.1, A 0, B 90, C -0, E1 0, E2 0, E3 0, E4 0} C_DIS
LIN {X 754.105, Y -453.848, Z 308.1, A 0, B 90, C -0, E1 0, E2 0, E3 0, E4 0} C_DIS
LIN {X 755.418, Y -455.454, Z 308.1, A 0, B 90, C -0, E1 0, E2 0, E3 0, E4 0} C_DIS
LIN {X 756.73, Y -457.059, Z 308.1, A 0, B 90, C -0, E1 0, E2 0, E3 0, E4 0} C_DIS
LIN {X 758.421, Y -458.105, Z 308.1, A 0, B 90, C -0, E1 0, E2 0, E3 0, E4 0} C_DIS
LIN {X 760.097, Y -456.973, Z 308.1, A 0, B 90, C -0, E1 0, E2 0, E3 0, E4 0} C_DIS
LIN {X 761.521, Y -455.465, Z 308.1, A 0, B 90, C -0, E1 0, E2 0, E3 0, E4 0} C_DIS
LIN {X 762.944, Y -453.957, Z 308.1, A 0, B 90, C -0, E1 0, E2 0, E3 0, E4 0} C_DIS
LIN {X 764.368, Y -452.449, Z 308.1, A 0, B 90, C -0, E1 0, E2 0, E3 0, E4 0} C_DIS
LIN {X 765.792, Y -450.941, Z 308.1, A 0, B 90, C -0, E1 0, E2 0, E3 0, E4 0} C_DIS
LIN {X 767.215, Y -449.433, Z 308.1, A 0, B 90, C -0, E1 0, E2 0, E3 0, E4 0} C_DIS
LIN {X 768.979, Y -448.412, Z 308.1, A 0, B 90, C -0, E1 0, E2 0, E3 0, E4 0} C_DIS
LIN {X 771, Y -448.719, Z 308.1, A 0, B 90, C -0, E1 0, E2 0, E3 0, E4 0} C_DIS
LIN {X 772.94, Y -449.453, Z 308.1, A 0, B 90, C -0, E1 0, E2 0, E3 0, E4 0} C_DIS
LIN {X 774.879, Y -450.187, Z 308.1, A 0, B 90, C -0, E1 0, E2 0, E3 0, E4 0} C_DIS
LIN {X 776.819, Y -450.921, Z 308.1, A 0, B 90, C -0, E1 0, E2 0, E3 0, E4 0} C_DIS
LIN {X 778.758, Y -451.655, Z 308.1, A 0, B 90, C -0, E1 0, E2 0, E3 0, E4 0} C_DIS
LIN {X 780.698, Y -452.389, Z 308.1, A 0, B 90, C -0, E1 0, E2 0, E3 0, E4 0} C_DIS
LIN {X 782.685, Y -452.45, Z 308.1, A 0, B 90, C -0, E1 0, E2 0, E3 0, E4 0} C_DIS
LIN {X 783.57, Y -450.631, Z 308.1, A 0, B 90, C -0, E1 0, E2 0, E3 0, E4 0} C_DIS
LIN {X 784.049, Y -448.613, Z 308.1, A 0, B 90, C -0, E1 0, E2 0, E3 0, E4 0} C_DIS
LIN {X 784.528, Y -446.596, Z 308.1, A 0, B 90, C -0, E1 0, E2 0, E3 0, E4 0} C_DIS
LIN {X 785.007, Y -444.578, Z 308.1, A 0, B 90, C -0, E1 0, E2 0, E3 0, E4 0} C_DIS
LIN {X 785.486, Y -442.56, Z 308.1, A 0, B 90, C -0, E1 0, E2 0, E3 0, E4 0} C_DIS
LIN {X 785.965, Y -440.542, Z 308.1, A 0, B 90, C -0, E1 0, E2 0, E3 0, E4 0} C_DIS
LIN {X 786.982, Y -438.776, Z 308.1, A 0, B 90, C -0, E1 0, E2 0, E3 0, E4 0} C_DIS
LIN {X 788.886, Y -438.031, Z 308.1, A 0, B 90, C -0, E1 0, E2 0, E3 0, E4 0} C_DIS
LIN {X 790.933, Y -437.697, Z 308.1, A 0, B 90, C -0, E1 0, E2 0, E3 0, E4 0} C_DIS
LIN {X 792.979, Y -437.363, Z 308.1, A 0, B 90, C -0, E1 0, E2 0, E3 0, E4 0} C_DIS
LIN {X 795.026, Y -437.029, Z 308.1, A 0, B 90, C -0, E1 0, E2 0, E3 0, E4 0} C_DIS
LIN {X 797.073, Y -436.695, Z 308.1, A 0, B 90, C -0, E1 0, E2 0, E3 0, E4 0} C_DIS
LIN {X 799.12, Y -436.361, Z 308.1, A 0, B 90, C -0, E1 0, E2 0, E3 0, E4 0} C_DIS
LIN {X 800.871, Y -435.42, Z 308.1, A 0, B 90, C -0, E1 0, E2 0, E3 0, E4 0} C_DIS
LIN {X 800.728, Y -433.403, Z 308.1, A 0, B 90, C -0, E1 0, E2 0, E3 0, E4 0} C_DIS
LIN {X 800.134, Y -431.416, Z 308.1, A 0, B 90, C -0, E1 0, E2 0, E3 0, E4 0} C_DIS
LIN {X 799.54, Y -429.429, Z 308.1, A 0, B 90, C -0, E1 0, E2 0, E3 0, E4 0} C_DIS
LIN {X 798.946, Y -427.442, Z 308.1, A 0, B 90, C -0, E1 0, E2 0, E3 0, E4 0} C_DIS
LIN {X 798.352, Y -425.455, Z 308.1, A 0, B 90, C -0, E1 0, E2 0, E3 0, E4 0} C_DIS
LIN {X 797.758, Y -423.468, Z 308.1, A 0, B 90, C -0, E1 0, E2 0, E3 0, E4 0} C_DIS
LIN {X 797.755, Y -421.43, Z 308.1, A 0, B 90, C -0, E1 0, E2 0, E3 0, E4 0} C_DIS
LIN {X 799.031, Y -419.833, Z 308.1, A 0, B 90, C -0, E1 0, E2 0, E3 0, E4 0} C_DIS
LIN {X 800.637, Y -418.52, Z 308.1, A 0, B 90, C -0, E1 0, E2 0, E3 0, E4 0} C_DIS
LIN {X 802.243, Y -417.208, Z 308.1, A 0, B 90, C -0, E1 0, E2 0, E3 0, E4 0} C_DIS
LIN {X 803.848, Y -415.895, Z 308.1, A 0, B 90, C -0, E1 0, E2 0, E3 0, E4 0} C_DIS
LIN {X 805.454, Y -414.582, Z 308.1, A 0, B 90, C -0, E1 0, E2 0, E3 0, E4 0} C_DIS
LIN {X 807.059, Y -413.27, Z 308.1, A 0, B 90, C -0, E1 0, E2 0, E3 0, E4 0} C_DIS
LIN {X 808.105, Y -411.579, Z 308.1, A 0, B 90, C -0, E1 0, E2 0, E3 0, E4 0} C_DIS
LIN {X 806.973, Y -409.903, Z 308.1, A 0, B 90, C -0, E1 0, E2 0, E3 0, E4 0} C_DIS
LIN {X 805.465, Y -408.48, Z 308.1, A 0, B 90, C -0, E1 0, E2 0, E3 0, E4 0} C_DIS
LIN {X 803.957, Y -407.056, Z 308.1, A 0, B 90, C -0, E1 0, E2 0, E3 0, E4 0} C_DIS
LIN {X 802.449, Y -405.632, Z 308.1, A 0, B 90, C -0, E1 0, E2 0, E3 0, E4 0} C_DIS
LIN {X 800.941, Y -404.208, Z 308.1, A 0, B 90, C -0, E1 0, E2 0, E3 0, E4 0} C_DIS
LIN {X 799.433, Y -402.785, Z 308.1, A 0, B 90, C -0, E1 0, E2 0, E3 0, E4 0} C_DIS
LIN {X 798.412, Y -401.021, Z 308.1, A 0, B 90, C -0, E1 0, E2 0, E3 0, E4 0} C_DIS
LIN {X 798.719, Y -399, Z 308.1, A 0, B 90, C -0, E1 0, E2 0, E3 0, E4 0} C_DIS
LIN {X 799.453, Y -397.06, Z 308.1, A 0, B 90, C -0, E1 0, E2 0, E3 0, E4 0} C_DIS
LIN {X 800.187, Y -395.121, Z 308.1, A 0, B 90, C -0, E1 0, E2 0, E3 0, E4 0} C_DIS
LIN {X 800.921, Y -393.181, Z 308.1, A 0, B 90, C -0, E1 0, E2 0, E3 0, E4 0} C_DIS
LIN {X 801.655, Y -391.242, Z 308.1, A 0, B 90, C -0, E1 0, E2 0, E3 0, E4 0} C_DIS
LIN {X 802.389, Y -389.302, Z 308.1, A 0, B 90, C -0, E1 0, E2 0, E3 0, E4 0} C_DIS
LIN {X 802.45, Y -387.315, Z 308.1, A 0, B 90, C -0, E1 0, E2 0, E3 0, E4 0} C_DIS
LIN {X 800.631, Y -386.43, Z 308.1, A 0, B 90, C -0, E1 0, E2 0, E3 0, E4 0} C_DIS
LIN {X 798.613, Y -385.951, Z 308.1, A 0, B 90, C -0, E1 0, E2 0, E3 0, E4 0} C_DIS
LIN {X 796.596, Y -385.472, Z 308.1, A 0, B 90, C -0, E1 0, E2 0, E3 0, E4 0} C_DIS
LIN {X 794.578, Y -384.993, Z 308.1, A 0, B 90, C -0, E1 0, E2 0, E3 0, E4 0} C_DIS
LIN {X 792.56, Y -384.514, Z 308.1, A 0, B 90, C -0, E1 0, E2 0, E3 0, E4 0} C_DIS
LIN {X 790.542, Y -384.035, Z 308.1, A 0, B 90, C -0, E1 0, E2 0, E3 0, E4 0} C_DIS
LIN {X 788.776, Y -383.018, Z 308.1, A 0, B 90, C -0, E1 0, E2 0, E3 0, E4 0} C_DIS
LIN {X 788.031, Y -381.114, Z 308.1, A 0, B 90, C -0, E1 0, E2 0, E3 0, E4 0} C_DIS
LIN {X 787.697, Y -379.067, Z 308.1, A 0, B 90, C -0, E1 0, E2 0, E3 0, E4 0} C_DIS
LIN {X 787.363, Y -377.021, Z 308.1, A 0, B 90, C -0, E1 0, E2 0, E3 0, E4 0} C_DIS
LIN {X 787.029, Y -374.974, Z 308.1, A 0, B 90, C -0, E1 0, E2 0, E3 0, E4 0} C_DIS
LIN {X 786.695, Y -372.927, Z 308.1, A 0, B 90, C -0, E1 0, E2 0, E3 0, E4 0} C_DIS
LIN {X 786.361, Y -370.88, Z 308.1, A 0, B 90, C -0, E1 0, E2 0, E3 0, E4 0} C_DIS
LIN {X 785.42, Y -369.129, Z 308.1, A 0, B 90, C -0, E1 0, E2 0, E3 0, E4 0} C_DIS
LIN {X 783.403, Y -369.272, Z 308.1, A 0, B 90, C -0, E1 0, E2 0, E3 0, E4 0} C_DIS
LIN {X 781.416, Y -369.866, Z 308.1, A 0, B 90, C -0, E1 0, E2 0, E3 0, E4 0} C_DIS
LIN {X 779.429, Y -370.46, Z 308.1, A 0, B 90, C -0, E1 0, E2 0, E3 0, E4 0} C_DIS
LIN {X 777.442, Y -371.054, Z 308.1, A 0, B 90, C -0, E1 0, E2 0, E3 0, E4 0} C_DIS
LIN {X 775.455, Y -371.648, Z 308.1, A 0, B 90, C -0, E1 0, E2 0, E3 0, E4 0} C_DIS
LIN {X 773.468, Y -372.242, Z 308.1, A 0, B 90, C -0, E1 0, E2 0, E3 0, E4 0} C_DIS
LIN {X 771.43, Y -372.245, Z 308.1, A 0, B 90, C -0, E1 0, E2 0, E3 0, E4 0} C_DIS
LIN {X 769.833, Y -370.969, Z 308.1, A 0, B 90, C -0, E1 0, E2 0, E3 0, E4 0} C_DIS
LIN {X 768.52, Y -369.363, Z 308.1, A 0, B 90, C -0, E1 0, E2 0, E3 0, E4 0} C_DIS
LIN {X 767.208, Y -367.757, Z 308.1, A 0, B 90, C -0, E1 0, E2 0, E3 0, E4 0} C_DIS
LIN {X 765.895, Y -366.152, Z 308.1, A 0, B 90, C -0, E1 0, E2 0, E3 0, E4 0} C_DIS
LIN {X 764.582, Y -364.546, Z 308.1, A 0, B 90, C -0, E1 0, E2 0, E3 0, E4 0} C_DIS
LIN {X 763.27, Y -362.941, Z 308.1, A 0, B 90, C -0, E1 0, E2 0, E3 0, E4 0} C_DIS
LIN {X 761.579, Y -361.895, Z 308.1, A 0, B 90, C -0, E1 0, E2 0, E3 0, E4 0} C_DIS
LIN {X 759.903, Y -363.027, Z 308.1, A 0, B 90, C -0, E1 0, E2 0, E3 0, E4 0} C_DIS
LIN {X 758.479, Y -364.535, Z 308.1, A 0, B 90, C -0, E1 0, E2 0, E3 0, E4 0} C_DIS
LIN {X 757.056, Y -366.043, Z 308.1, A 0, B 90, C -0, E1 0, E2 0, E3 0, E4 0} C_DIS
LIN {X 755.632, Y -367.551, Z 308.1, A 0, B 90, C -0, E1 0, E2 0, E3 0, E4 0} C_DIS
LIN {X 754.208, Y -369.059, Z 308.1, A 0, B 90, C -0, E1 0, E2 0, E3 0, E4 0} C_DIS
LIN {X 752.674, Y -370.587, Z 309.4, A 0, B 90, C -0, E1 0, E2 0, E3 0, E4 0} C_DIS
LIN {X 750.914, Y -371.613, Z 309.4, A 0, B 90, C -0, E1 0, E2 0, E3 0, E4 0} C_DIS
LIN {X 748.891, Y -371.312, Z 309.4, A 0, B 90, C -0, E1 0, E2 0, E3 0, E4 0} C_DIS
LIN {X 746.949, Y -370.583, Z 309.4, A 0, B 90, C -0, E1 0, E2 0, E3 0, E4 0} C_DIS
LIN {X 745.008, Y -369.854, Z 309.4, A 0, B 90, C -0, E1 0, E2 0, E3 0, E4 0} C_DIS
LIN {X 743.066, Y -369.125, Z 309.4, A 0, B 90, C -0, E1 0, E2 0, E3 0, E4 0} C_DIS
LIN {X 741.124, Y -368.397, Z 309.4, A 0, B 90, C -0, E1 0, E2 0, E3 0, E4 0} C_DIS
LIN {X 739.183, Y -367.668, Z 309.4, A 0, B 90, C -0, E1 0, E2 0, E3 0, E4 0} C_DIS
LIN {X 737.195, Y -367.613, Z 309.4, A 0, B 90, C -0, E1 0, E2 0, E3 0, E4 0} C_DIS
LIN {X 736.315, Y -369.434, Z 309.4, A 0, B 90, C -0, E1 0, E2 0, E3 0, E4 0} C_DIS
LIN {X 735.842, Y -371.453, Z 309.4, A 0, B 90, C -0, E1 0, E2 0, E3 0, E4 0} C_DIS
LIN {X 735.369, Y -373.472, Z 309.4, A 0, B 90, C -0, E1 0, E2 0, E3 0, E4 0} C_DIS
LIN {X 734.895, Y -375.492, Z 309.4, A 0, B 90, C -0, E1 0, E2 0, E3 0, E4 0} C_DIS
LIN {X 734.422, Y -377.511, Z 309.4, A 0, B 90, C -0, E1 0, E2 0, E3 0, E4 0} C_DIS
LIN {X 733.949, Y -379.53, Z 309.4, A 0, B 90, C -0, E1 0, E2 0, E3 0, E4 0} C_DIS
LIN {X 732.937, Y -381.299, Z 309.4, A 0, B 90, C -0, E1 0, E2 0, E3 0, E4 0} C_DIS
LIN {X 731.035, Y -382.049, Z 309.4, A 0, B 90, C -0, E1 0, E2 0, E3 0, E4 0} C_DIS
LIN {X 728.989, Y -382.389, Z 309.4, A 0, B 90, C -0, E1 0, E2 0, E3 0, E4 0} C_DIS
LIN {X 726.943, Y -382.729, Z 309.4, A 0, B 90, C -0, E1 0, E2 0, E3 0, E4 0} C_DIS
LIN {X 724.897, Y -383.068, Z 309.4, A 0, B 90, C -0, E1 0, E2 0, E3 0, E4 0} C_DIS
LIN {X 722.851, Y -383.408, Z 309.4, A 0, B 90, C -0, E1 0, E2 0, E3 0, E4 0} C_DIS
LIN {X 720.806, Y -383.748, Z 309.4, A 0, B 90, C -0, E1 0, E2 0, E3 0, E4 0} C_DIS
LIN {X 719.057, Y -384.694, Z 309.4, A 0, B 90, C -0, E1 0, E2 0, E3 0, E4 0} C_DIS
LIN {X 719.206, Y -386.711, Z 309.4, A 0, B 90, C -0, E1 0, E2 0, E3 0, E4 0} C_DIS
LIN {X 719.805, Y -388.697, Z 309.4, A 0, B 90, C -0, E1 0, E2 0, E3 0, E4 0} C_DIS
LIN {X 720.405, Y -390.682, Z 309.4, A 0, B 90, C -0, E1 0, E2 0, E3 0, E4 0} C_DIS
LIN {X 721.005, Y -392.667, Z 309.4, A 0, B 90, C -0, E1 0, E2 0, E3 0, E4 0} C_DIS
LIN {X 721.604, Y -394.652, Z 309.4, A 0, B 90, C -0, E1 0, E2 0, E3 0, E4 0} C_DIS
LIN {X 722.204, Y -396.638, Z 309.4, A 0, B 90, C -0, E1 0, E2 0, E3 0, E4 0} C_DIS
LIN {X 722.212, Y -398.676, Z 309.4, A 0, B 90, C -0, E1 0, E2 0, E3 0, E4 0} C_DIS
LIN {X 720.94, Y -400.277, Z 309.4, A 0, B 90, C -0, E1 0, E2 0, E3 0, E4 0} C_DIS
LIN {X 719.338, Y -401.594, Z 309.4, A 0, B 90, C -0, E1 0, E2 0, E3 0, E4 0} C_DIS
LIN {X 717.736, Y -402.911, Z 309.4, A 0, B 90, C -0, E1 0, E2 0, E3 0, E4 0} C_DIS
LIN {X 716.134, Y -404.228, Z 309.4, A 0, B 90, C -0, E1 0, E2 0, E3 0, E4 0} C_DIS
LIN {X 714.533, Y -405.545, Z 309.4, A 0, B 90, C -0, E1 0, E2 0, E3 0, E4 0} C_DIS
LIN {X 712.931, Y -406.862, Z 309.4, A 0, B 90, C -0, E1 0, E2 0, E3 0, E4 0} C_DIS
LIN {X 711.89, Y -408.556, Z 309.4, A 0, B 90, C -0, E1 0, E2 0, E3 0, E4 0} C_DIS
LIN {X 713.027, Y -410.229, Z 309.4, A 0, B 90, C -0, E1 0, E2 0, E3 0, E4 0} C_DIS
LIN {X 714.539, Y -411.648, Z 309.4, A 0, B 90, C -0, E1 0, E2 0, E3 0, E4 0} C_DIS
LIN {X 716.051, Y -413.068, Z 309.4, A 0, B 90, C -0, E1 0, E2 0, E3 0, E4 0} C_DIS
LIN {X 717.563, Y -414.487, Z 309.4, A 0, B 90, C -0, E1 0, E2 0, E3 0, E4 0} C_DIS
LIN {X 719.075, Y -415.906, Z 309.4, A 0, B 90, C -0, E1 0, E2 0, E3 0, E4 0} C_DIS
LIN {X 720.587, Y -417.326, Z 309.4, A 0, B 90, C -0, E1 0, E2 0, E3 0, E4 0} C_DIS
LIN {X 721.613, Y -419.087, Z 309.4, A 0, B 90, C -0, E1 0, E2 0, E3 0, E4 0} C_DIS
LIN {X 721.312, Y -421.109, Z 309.4, A 0, B 90, C -0, E1 0, E2 0, E3 0, E4 0} C_DIS
LIN {X 720.583, Y -423.051, Z 309.4, A 0, B 90, C -0, E1 0, E2 0, E3 0, E4 0} C_DIS
LIN {X 719.854, Y -424.992, Z 309.4, A 0, B 90, C -0, E1 0, E2 0, E3 0, E4 0} C_DIS
LIN {X 719.125, Y -426.934, Z 309.4, A 0, B 90, C -0, E1 0, E2 0, E3 0, E4 0} C_DIS
LIN {X 718.397, Y -428.876, Z 309.4, A 0, B 90, C -0, E1 0, E2 0, E3 0, E4 0} C_DIS
LIN {X 717.668, Y -430.817, Z 309.4, A 0, B 90, C -0, E1 0, E2 0, E3 0, E4 0} C_DIS
LIN {X 717.613, Y -432.805, Z 309.4, A 0, B 90, C -0, E1 0, E2 0, E3 0, E4 0} C_DIS
LIN {X 719.434, Y -433.685, Z 309.4, A 0, B 90, C -0, E1 0, E2 0, E3 0, E4 0} C_DIS
LIN {X 721.453, Y -434.158, Z 309.4, A 0, B 90, C -0, E1 0, E2 0, E3 0, E4 0} C_DIS
LIN {X 723.472, Y -434.631, Z 309.4, A 0, B 90, C -0, E1 0, E2 0, E3 0, E4 0} C_DIS
LIN {X 725.492, Y -435.105, Z 309.4, A 0, B 90, C -0, E1 0, E2 0, E3 0, E4 0} C_DIS
LIN {X 727.511, Y -435.578, Z 309.4, A 0, B 90, C -0, E1 0, E2 0, E3 0, E4 0} C_DIS
LIN {X 729.53, Y -436.051, Z 309.4, A 0, B 90, C -0, E1 0, E2 0, E3 0, E4 0} C_DIS
LIN {X 731.299, Y -437.063, Z 309.4, A 0, B 90, C -0, E1 0, E2 0, E3 0, E4 0} C_DIS
LIN {X 732.049, Y -438.965, Z 309.4, A 0, B 90, C -0, E1 0, E2 0, E3 0, E4 0} C_DIS
LIN {X 732.389, Y -441.011, Z 309.4, A 0, B 90, C -0, E1 0, E2 0, E3 0, E4 0} C_DIS
LIN {X 732.729, Y -443.057, Z 309.4, A 0, B 90, C -0, E1 0, E2 0, E3 0, E4 0} C_DIS
LIN {X 733.068, Y -445.103, Z 309.4, A 0, B 90, C -0, E1 0, E2 0, E3 0, E4 0} C_DIS
LIN {X 733.408, Y -447.149, Z 309.4, A 0, B 90, C -0, E1 0, E2 0, E3 0, E4 0} C_DIS
LIN {X 733.748, Y -449.194, Z 309.4, A 0, B 90, C -0, E1 0, E2 0, E3 0, E4 0} C_DIS
LIN {X 734.694, Y -450.943, Z 309.4, A 0, B 90, C -0, E1 0, E2 0, E3 0, E4 0} C_DIS
LIN {X 736.711, Y -450.794, Z 309.4, A 0, B 90, C -0, E1 0, E2 0, E3 0, E4 0} C_DIS
LIN {X 738.697, Y -450.195, Z 309.4, A 0, B 90, C -0, E1 0, E2 0, E3 0, E4 0} C_DIS
LIN {X 740.682, Y -449.595, Z 309.4, A 0, B 90, C -0, E1 0, E2 0, E3 0, E4 0} C_DIS
LIN {X 742.667, Y -448.995, Z 309.4, A 0, B 90, C -0, E1 0, E2 0, E3 0, E4 0} C_DIS
LIN {X 744.652, Y -448.396, Z 309.4, A 0, B 90, C -0, E1 0, E2 0, E3 0, E4 0} C_DIS
LIN {X 746.638, Y -447.796, Z 309.4, A 0, B 90, C -0, E1 0, E2 0, E3 0, E4 0} C_DIS
LIN {X 748.676, Y -447.788, Z 309.4, A 0, B 90, C -0, E1 0, E2 0, E3 0, E4 0} C_DIS
LIN {X 750.277, Y -449.06, Z 309.4, A 0, B 90, C -0, E1 0, E2 0, E3 0, E4 0} C_DIS
LIN {X 751.594, Y -450.662, Z 309.4, A 0, B 90, C -0, E1 0, E2 0, E3 0, E4 0} C_DIS
LIN {X 752.911, Y -452.264, Z 309.4, A 0, B 90, C -0, E1 0, E2 0, E3 0, E4 0} C_DIS
LIN {X 754.228, Y -453.866, Z 309.4, A 0, B 90, C -0, E1 0, E2 0, E3 0, E4 0} C_DIS
LIN {X 755.545, Y -455.467, Z 309.4, A 0, B 90, C -0, E1 0, E2 0, E3 0, E4 0} C_DIS
LIN {X 756.862, Y -457.069, Z 309.4, A 0, B 90, C -0, E1 0, E2 0, E3 0, E4 0} C_DIS
LIN {X 758.556, Y -458.11, Z 309.4, A 0, B 90, C -0, E1 0, E2 0, E3 0, E4 0} C_DIS
LIN {X 760.229, Y -456.973, Z 309.4, A 0, B 90, C -0, E1 0, E2 0, E3 0, E4 0} C_DIS
LIN {X 761.648, Y -455.461, Z 309.4, A 0, B 90, C -0, E1 0, E2 0, E3 0, E4 0} C_DIS
LIN {X 763.068, Y -453.949, Z 309.4, A 0, B 90, C -0, E1 0, E2 0, E3 0, E4 0} C_DIS
LIN {X 764.487, Y -452.437, Z 309.4, A 0, B 90, C -0, E1 0, E2 0, E3 0, E4 0} C_DIS
LIN {X 765.906, Y -450.925, Z 309.4, A 0, B 90, C -0, E1 0, E2 0, E3 0, E4 0} C_DIS
LIN {X 767.326, Y -449.413, Z 309.4, A 0, B 90, C -0, E1 0, E2 0, E3 0, E4 0} C_DIS
LIN {X 769.086, Y -448.387, Z 309.4, A 0, B 90, C -0, E1 0, E2 0, E3 0, E4 0} C_DIS
LIN {X 771.109, Y -448.688, Z 309.4, A 0, B 90, C -0, E1 0, E2 0, E3 0, E4 0} C_DIS
LIN {X 773.051, Y -449.417, Z 309.4, A 0, B 90, C -0, E1 0, E2 0, E3 0, E4 0} C_DIS
LIN {X 774.992, Y -450.146, Z 309.4, A 0, B 90, C -0, E1 0, E2 0, E3 0, E4 0} C_DIS
LIN {X 776.934, Y -450.875, Z 309.4, A 0, B 90, C -0, E1 0, E2 0, E3 0, E4 0} C_DIS
LIN {X 778.876, Y -451.603, Z 309.4, A 0, B 90, C -0, E1 0, E2 0, E3 0, E4 0} C_DIS
LIN {X 780.817, Y -452.332, Z 309.4, A 0, B 90, C -0, E1 0, E2 0, E3 0, E4 0} C_DIS
LIN {X 782.805, Y -452.387, Z 309.4, A 0, B 90, C -0, E1 0, E2 0, E3 0, E4 0} C_DIS
LIN {X 783.685, Y -450.566, Z 309.4, A 0, B 90, C -0, E1 0, E2 0, E3 0, E4 0} C_DIS
LIN {X 784.158, Y -448.547, Z 309.4, A 0, B 90, C -0, E1 0, E2 0, E3 0, E4 0} C_DIS
LIN {X 784.631, Y -446.528, Z 309.4, A 0, B 90, C -0, E1 0, E2 0, E3 0, E4 0} C_DIS
LIN {X 785.105, Y -444.508, Z 309.4, A 0, B 90, C -0, E1 0, E2 0, E3 0, E4 0} C_DIS
LIN {X 785.578, Y -442.489, Z 309.4, A 0, B 90, C -0, E1 0, E2 0, E3 0, E4 0} C_DIS
LIN {X 786.051, Y -440.47, Z 309.4, A 0, B 90, C -0, E1 0, E2 0, E3 0, E4 0} C_DIS
LIN {X 787.063, Y -438.701, Z 309.4, A 0, B 90, C -0, E1 0, E2 0, E3 0, E4 0} C_DIS
LIN {X 788.965, Y -437.951, Z 309.4, A 0, B 90, C -0, E1 0, E2 0, E3 0, E4 0} C_DIS
LIN {X 791.011, Y -437.611, Z 309.4, A 0, B 90, C -0, E1 0, E2 0, E3 0, E4 0} C_DIS
LIN {X 793.057, Y -437.271, Z 309.4, A 0, B 90, C -0, E1 0, E2 0, E3 0, E4 0} C_DIS
LIN {X 795.103, Y -436.932, Z 309.4, A 0, B 90, C -0, E1 0, E2 0, E3 0, E4 0} C_DIS
LIN {X 797.149, Y -436.592, Z 309.4, A 0, B 90, C -0, E1 0, E2 0, E3 0, E4 0} C_DIS
LIN {X 799.194, Y -436.252, Z 309.4, A 0, B 90, C -0, E1 0, E2 0, E3 0, E4 0} C_DIS
LIN {X 800.943, Y -435.306, Z 309.4, A 0, B 90, C -0, E1 0, E2 0, E3 0, E4 0} C_DIS
LIN {X 800.794, Y -433.289, Z 309.4, A 0, B 90, C -0, E1 0, E2 0, E3 0, E4 0} C_DIS
LIN {X 800.195, Y -431.303, Z 309.4, A 0, B 90, C -0, E1 0, E2 0, E3 0, E4 0} C_DIS
LIN {X 799.595, Y -429.318, Z 309.4, A 0, B 90, C -0, E1 0, E2 0, E3 0, E4 0} C_DIS
LIN {X 798.995, Y -427.333, Z 309.4, A 0, B 90, C -0, E1 0, E2 0, E3 0, E4 0} C_DIS
LIN {X 798.396, Y -425.348, Z 309.4, A 0, B 90, C -0, E1 0, E2 0, E3 0, E4 0} C_DIS
LIN {X 797.796, Y -423.362, Z 309.4, A 0, B 90, C -0, E1 0, E2 0, E3 0, E4 0} C_DIS
LIN {X 797.788, Y -421.324, Z 309.4, A 0, B 90, C -0, E1 0, E2 0, E3 0, E4 0} C_DIS
LIN {X 799.06, Y -419.723, Z 309.4, A 0, B 90, C -0, E1 0, E2 0, E3 0, E4 0} C_DIS
LIN {X 800.662, Y -418.406, Z 309.4, A 0, B 90, C -0, E1 0, E2 0, E3 0, E4 0} C_DIS
LIN {X 802.264, Y -417.089, Z 309.4, A 0, B 90, C -0, E1 0, E2 0, E3 0, E4 0} C_DIS
LIN {X 803.866, Y -415.772, Z 309.4, A 0, B 90, C -0, E1 0, E2 0, E3 0, E4 0} C_DIS
LIN {X 805.467, Y -414.455, Z 309.4, A 0, B 90, C -0, E1 0, E2 0, E3 0, E4 0} C_DIS
LIN {X 807.069, Y -413.138, Z 309.4, A 0, B 90, C -0, E1 0, E2 0, E3 0, E4 0} C_DIS
LIN {X 808.11, Y -411.444, Z 309.4, A 0, B 90, C -0, E1 0, E2 0, E3 0, E4 0} C_DIS
LIN {X 806.973, Y -409.771, Z 309.4, A 0, B 90, C -0, E1 0, E2 0, E3 0, E4 0} C_DIS
LIN {X 805.461, Y -408.352, Z 309.4, A 0, B 90, C -0, E1 0, E2 0, E3 0, E4 0} C_DIS
LIN {X 803.949, Y -406.932, Z 309.4, A 0, B 90, C -0, E1 0, E2 0, E3 0, E4 0} C_DIS
LIN {X 802.437, Y -405.513, Z 309.4, A 0, B 90, C -0, E1 0, E2 0, E3 0, E4 0} C_DIS
LIN {X 800.925, Y -404.094, Z 309.4, A 0, B 90, C -0, E1 0, E2 0, E3 0, E4 0} C_DIS
LIN {X 799.413, Y -402.674, Z 309.4, A 0, B 90, C -0, E1 0, E2 0, E3 0, E4 0} C_DIS
LIN {X 798.387, Y -400.913, Z 309.4, A 0, B 90, C -0, E1 0, E2 0, E3 0, E4 0} C_DIS
LIN {X 798.688, Y -398.891, Z 309.4, A 0, B 90, C -0, E1 0, E2 0, E3 0, E4 0} C_DIS
LIN {X 799.417, Y -396.949, Z 309.4, A 0, B 90, C -0, E1 0, E2 0, E3 0, E4 0} C_DIS
LIN {X 800.146, Y -395.008, Z 309.4, A 0, B 90, C -0, E1 0, E2 0, E3 0, E4 0} C_DIS
LIN {X 800.875, Y -393.066, Z 309.4, A 0, B 90, C -0, E1 0, E2 0, E3 0, E4 0} C_DIS
LIN {X 801.603, Y -391.124, Z 309.4, A 0, B 90, C -0, E1 0, E2 0, E3 0, E4 0} C_DIS
LIN {X 802.332, Y -389.183, Z 309.4, A 0, B 90, C -0, E1 0, E2 0, E3 0, E4 0} C_DIS
LIN {X 802.387, Y -387.195, Z 309.4, A 0, B 90, C -0, E1 0, E2 0, E3 0, E4 0} C_DIS
LIN {X 800.566, Y -386.315, Z 309.4, A 0, B 90, C -0, E1 0, E2 0, E3 0, E4 0} C_DIS
LIN {X 798.547, Y -385.842, Z 309.4, A 0, B 90, C -0, E1 0, E2 0, E3 0, E4 0} C_DIS
LIN {X 796.528, Y -385.369, Z 309.4, A 0, B 90, C -0, E1 0, E2 0, E3 0, E4 0} C_DIS
LIN {X 794.508, Y -384.895, Z 309.4, A 0, B 90, C -0, E1 0, E2 0, E3 0, E4 0} C_DIS
LIN {X 792.489, Y -384.422, Z 309.4, A 0, B 90, C -0, E1 0, E2 0, E3 0, E4 0} C_DIS
LIN {X 790.47, Y -383.949, Z 309.4, A 0, B 90, C -0, E1 0, E2 0, E3 0, E4 0} C_DIS
LIN {X 788.701, Y -382.937, Z 309.4, A 0, B 90, C -0, E1 0, E2 0, E3 0, E4 0} C_DIS
LIN {X 787.951, Y -381.035, Z 309.4, A 0, B 90, C -0, E1 0, E2 0, E3 0, E4 0} C_DIS
LIN {X 787.611, Y -378.989, Z 309.4, A 0, B 90, C -0, E1 0, E2 0, E3 0, E4 0} C_DIS
LIN {X 787.271, Y -376.943, Z 309.4, A 0, B 90, C -0, E1 0, E2 0, E3 0, E4 0} C_DIS
LIN {X 786.932, Y -374.897, Z 309.4, A 0, B 90, C -0, E1 0, E2 0, E3 0, E4 0} C_DIS
LIN {X 786.592, Y -372.851, Z 309.4, A 0, B 90, C -0, E1 0, E2 0, E3 0, E4 0} C_DIS
LIN {X 786.252, Y -370.806, Z 309.4, A 0, B 90, C -0, E1 0, E2 0, E3 0, E4 0} C_DIS
LIN {X 785.306, Y -369.057, Z 309.4, A 0, B 90, C -0, E1 0, E2 0, E3 0, E4 0} C_DIS
LIN {X 783.289, Y -369.206, Z 309.4, A 0, B 90, C -0, E1 0, E2 0, E3 0, E4 0} C_DIS
LIN {X 781.303, Y -369.805, Z 309.4, A 0, B 90, C -0, E1 0, E2 0, E3 0, E4 0} C_DIS
LIN {X 779.318, Y -370.405, Z 309.4, A 0, B 90, C -0, E1 0, E2 0, E3 0, E4 0} C_DIS
LIN {X 777.333, Y -371.005, Z 309.4, A 0, B 90, C -0, E1 0, E2 0, E3 0, E4 0} C_DIS
LIN {X 775.348, Y -371.604, Z 309.4, A 0, B 90, C -0, E1 0, E2 0, E3 0, E4 0} C_DIS
LIN {X 773.362, Y -372.204, Z 309.4, A 0, B 90, C -0, E1 0, E2 0, E3 0, E4 0} C_DIS
LIN {X 771.324, Y -372.212, Z 309.4, A 0, B 90, C -0, E1 0, E2 0, E3 0, E4 0} C_DIS
LIN {X 769.723, Y -370.94, Z 309.4, A 0, B 90, C -0, E1 0, E2 0, E3 0, E4 0} C_DIS
LIN {X 768.406, Y -369.338, Z 309.4, A 0, B 90, C -0, E1 0, E2 0, E3 0, E4 0} C_DIS
LIN {X 767.089, Y -367.736, Z 309.4, A 0, B 90, C -0, E1 0, E2 0, E3 0, E4 0} C_DIS
LIN {X 765.772, Y -366.134, Z 309.4, A 0, B 90, C -0, E1 0, E2 0, E3 0, E4 0} C_DIS
LIN {X 764.455, Y -364.533, Z 309.4, A 0, B 90, C -0, E1 0, E2 0, E3 0, E4 0} C_DIS
LIN {X 763.138, Y -362.931, Z 309.4, A 0, B 90, C -0, E1 0, E2 0, E3 0, E4 0} C_DIS
LIN {X 761.444, Y -361.89, Z 309.4, A 0, B 90, C -0, E1 0, E2 0, E3 0, E4 0} C_DIS
LIN {X 759.771, Y -363.027, Z 309.4, A 0, B 90, C -0, E1 0, E2 0, E3 0, E4 0} C_DIS
LIN {X 758.352, Y -364.539, Z 309.4, A 0, B 90, C -0, E1 0, E2 0, E3 0, E4 0} C_DIS
LIN {X 756.932, Y -366.051, Z 309.4, A 0, B 90, C -0, E1 0, E2 0, E3 0, E4 0} C_DIS
LIN {X 755.513, Y -367.563, Z 309.4, A 0, B 90, C -0, E1 0, E2 0, E3 0, E4 0} C_DIS
LIN {X 754.094, Y -369.075, Z 309.4, A 0, B 90, C -0, E1 0, E2 0, E3 0, E4 0} C_DIS
LIN {X 752.567, Y -370.603, Z 310.7, A 0, B 90, C -0, E1 0, E2 0, E3 0, E4 0} C_DIS
LIN {X 750.809, Y -371.634, Z 310.7, A 0, B 90, C -0, E1 0, E2 0, E3 0, E4 0} C_DIS
LIN {X 748.785, Y -371.338, Z 310.7, A 0, B 90, C -0, E1 0, E2 0, E3 0, E4 0} C_DIS
LIN {X 746.842, Y -370.614, Z 310.7, A 0, B 90, C -0, E1 0, E2 0, E3 0, E4 0} C_DIS
LIN {X 744.898, Y -369.891, Z 310.7, A 0, B 90, C -0, E1 0, E2 0, E3 0, E4 0} C_DIS
LIN {X 742.954, Y -369.167, Z 310.7, A 0, B 90, C -0, E1 0, E2 0, E3 0, E4 0} C_DIS
LIN {X 741.01, Y -368.444, Z 310.7, A 0, B 90, C -0, E1 0, E2 0, E3 0, E4 0} C_DIS
LIN {X 739.067, Y -367.72, Z 310.7, A 0, B 90, C -0, E1 0, E2 0, E3 0, E4 0} C_DIS
LIN {X 737.079, Y -367.671, Z 310.7, A 0, B 90, C -0, E1 0, E2 0, E3 0, E4 0} C_DIS
LIN {X 736.204, Y -369.494, Z 310.7, A 0, B 90, C -0, E1 0, E2 0, E3 0, E4 0} C_DIS
LIN {X 735.736, Y -371.515, Z 310.7, A 0, B 90, C -0, E1 0, E2 0, E3 0, E4 0} C_DIS
LIN {X 735.268, Y -373.535, Z 310.7, A 0, B 90, C -0, E1 0, E2 0, E3 0, E4 0} C_DIS
LIN {X 734.8, Y -375.556, Z 310.7, A 0, B 90, C -0, E1 0, E2 0, E3 0, E4 0} C_DIS
LIN {X 734.332, Y -377.577, Z 310.7, A 0, B 90, C -0, E1 0, E2 0, E3 0, E4 0} C_DIS
LIN {X 733.864, Y -379.597, Z 310.7, A 0, B 90, C -0, E1 0, E2 0, E3 0, E4 0} C_DIS
LIN {X 732.857, Y -381.369, Z 310.7, A 0, B 90, C -0, E1 0, E2 0, E3 0, E4 0} C_DIS
LIN {X 730.957, Y -382.125, Z 310.7, A 0, B 90, C -0, E1 0, E2 0, E3 0, E4 0} C_DIS
LIN {X 728.912, Y -382.47, Z 310.7, A 0, B 90, C -0, E1 0, E2 0, E3 0, E4 0} C_DIS
LIN {X 726.867, Y -382.815, Z 310.7, A 0, B 90, C -0, E1 0, E2 0, E3 0, E4 0} C_DIS
LIN {X 724.821, Y -383.161, Z 310.7, A 0, B 90, C -0, E1 0, E2 0, E3 0, E4 0} C_DIS
LIN {X 722.776, Y -383.506, Z 310.7, A 0, B 90, C -0, E1 0, E2 0, E3 0, E4 0} C_DIS
LIN {X 720.731, Y -383.851, Z 310.7, A 0, B 90, C -0, E1 0, E2 0, E3 0, E4 0} C_DIS
LIN {X 718.985, Y -384.802, Z 310.7, A 0, B 90, C -0, E1 0, E2 0, E3 0, E4 0} C_DIS
LIN {X 719.139, Y -386.819, Z 310.7, A 0, B 90, C -0, E1 0, E2 0, E3 0, E4 0} C_DIS
LIN {X 719.744, Y -388.803, Z 310.7, A 0, B 90, C -0, E1 0, E2 0, E3 0, E4 0} C_DIS
LIN {X 720.349, Y -390.787, Z 310.7, A 0, B 90, C -0, E1 0, E2 0, E3 0, E4 0} C_DIS
LIN {X 720.954, Y -392.771, Z 310.7, A 0, B 90, C -0, E1 0, E2 0, E3 0, E4 0} C_DIS
LIN {X 721.559, Y -394.755, Z 310.7, A 0, B 90, C -0, E1 0, E2 0, E3 0, E4 0} C_DIS
LIN {X 722.164, Y -396.738, Z 310.7, A 0, B 90, C -0, E1 0, E2 0, E3 0, E4 0} C_DIS
LIN {X 722.178, Y -398.776, Z 310.7, A 0, B 90, C -0, E1 0, E2 0, E3 0, E4 0} C_DIS
LIN {X 720.91, Y -400.381, Z 310.7, A 0, B 90, C -0, E1 0, E2 0, E3 0, E4 0} C_DIS
LIN {X 719.312, Y -401.703, Z 310.7, A 0, B 90, C -0, E1 0, E2 0, E3 0, E4 0} C_DIS
LIN {X 717.713, Y -403.024, Z 310.7, A 0, B 90, C -0, E1 0, E2 0, E3 0, E4 0} C_DIS
LIN {X 716.115, Y -404.346, Z 310.7, A 0, B 90, C -0, E1 0, E2 0, E3 0, E4 0} C_DIS
LIN {X 714.516, Y -405.667, Z 310.7, A 0, B 90, C -0, E1 0, E2 0, E3 0, E4 0} C_DIS
LIN {X 712.918, Y -406.989, Z 310.7, A 0, B 90, C -0, E1 0, E2 0, E3 0, E4 0} C_DIS
LIN {X 711.881, Y -408.686, Z 310.7, A 0, B 90, C -0, E1 0, E2 0, E3 0, E4 0} C_DIS
LIN {X 713.023, Y -410.355, Z 310.7, A 0, B 90, C -0, E1 0, E2 0, E3 0, E4 0} C_DIS
LIN {X 714.539, Y -411.771, Z 310.7, A 0, B 90, C -0, E1 0, E2 0, E3 0, E4 0} C_DIS
LIN {X 716.055, Y -413.186, Z 310.7, A 0, B 90, C -0, E1 0, E2 0, E3 0, E4 0} C_DIS
LIN {X 717.571, Y -414.602, Z 310.7, A 0, B 90, C -0, E1 0, E2 0, E3 0, E4 0} C_DIS
LIN {X 719.087, Y -416.017, Z 310.7, A 0, B 90, C -0, E1 0, E2 0, E3 0, E4 0} C_DIS
LIN {X 720.603, Y -417.433, Z 310.7, A 0, B 90, C -0, E1 0, E2 0, E3 0, E4 0} C_DIS
LIN {X 721.634, Y -419.191, Z 310.7, A 0, B 90, C -0, E1 0, E2 0, E3 0, E4 0} C_DIS
LIN {X 721.338, Y -421.215, Z 310.7, A 0, B 90, C -0, E1 0, E2 0, E3 0, E4 0} C_DIS
LIN {X 720.614, Y -423.158, Z 310.7, A 0, B 90, C -0, E1 0, E2 0, E3 0, E4 0} C_DIS
LIN {X 719.891, Y -425.102, Z 310.7, A 0, B 90, C -0, E1 0, E2 0, E3 0, E4 0} C_DIS
LIN {X 719.167, Y -427.046, Z 310.7, A 0, B 90, C -0, E1 0, E2 0, E3 0, E4 0} C_DIS
LIN {X 718.444, Y -428.99, Z 310.7, A 0, B 90, C -0, E1 0, E2 0, E3 0, E4 0} C_DIS
LIN {X 717.72, Y -430.933, Z 310.7, A 0, B 90, C -0, E1 0, E2 0, E3 0, E4 0} C_DIS
LIN {X 717.671, Y -432.921, Z 310.7, A 0, B 90, C -0, E1 0, E2 0, E3 0, E4 0} C_DIS
LIN {X 719.494, Y -433.796, Z 310.7, A 0, B 90, C -0, E1 0, E2 0, E3 0, E4 0} C_DIS
LIN {X 721.515, Y -434.264, Z 310.7, A 0, B 90, C -0, E1 0, E2 0, E3 0, E4 0} C_DIS
LIN {X 723.535, Y -434.732, Z 310.7, A 0, B 90, C -0, E1 0, E2 0, E3 0, E4 0} C_DIS
LIN {X 725.556, Y -435.2, Z 310.7, A 0, B 90, C -0, E1 0, E2 0, E3 0, E4 0} C_DIS
LIN {X 727.577, Y -435.668, Z 310.7, A 0, B 90, C -0, E1 0, E2 0, E3 0, E4 0} C_DIS
LIN {X 729.597, Y -436.136, Z 310.7, A 0, B 90, C -0, E1 0, E2 0, E3 0, E4 0} C_DIS
LIN {X 731.369, Y -437.143, Z 310.7, A 0, B 90, C -0, E1 0, E2 0, E3 0, E4 0} C_DIS
LIN {X 732.125, Y -439.043, Z 310.7, A 0, B 90, C -0, E1 0, E2 0, E3 0, E4 0} C_DIS
LIN {X 732.47, Y -441.088, Z 310.7, A 0, B 90, C -0, E1 0, E2 0, E3 0, E4 0} C_DIS
LIN {X 732.815, Y -443.133, Z 310.7, A 0, B 90, C -0, E1 0, E2 0, E3 0, E4 0} C_DIS
LIN {X 733.161, Y -445.179, Z 310.7, A 0, B 90, C -0, E1 0, E2 0, E3 0, E4 0} C_DIS
LIN {X 733.506, Y -447.224, Z 310.7, A 0, B 90, C -0, E1 0, E2 0, E3 0, E4 0} C_DIS
LIN {X 733.851, Y -449.269, Z 310.7, A 0, B 90, C -0, E1 0, E2 0, E3 0, E4 0} C_DIS
LIN {X 734.802, Y -451.015, Z 310.7, A 0, B 90, C -0, E1 0, E2 0, E3 0, E4 0} C_DIS
LIN {X 736.819, Y -450.861, Z 310.7, A 0, B 90, C -0, E1 0, E2 0, E3 0, E4 0} C_DIS
LIN {X 738.803, Y -450.256, Z 310.7, A 0, B 90, C -0, E1 0, E2 0, E3 0, E4 0} C_DIS
LIN {X 740.787, Y -449.651, Z 310.7, A 0, B 90, C -0, E1 0, E2 0, E3 0, E4 0} C_DIS
LIN {X 742.771, Y -449.046, Z 310.7, A 0, B 90, C -0, E1 0, E2 0, E3 0, E4 0} C_DIS
LIN {X 744.755, Y -448.441, Z 310.7, A 0, B 90, C -0, E1 0, E2 0, E3 0, E4 0} C_DIS
LIN {X 746.738, Y -447.836, Z 310.7, A 0, B 90, C -0, E1 0, E2 0, E3 0, E4 0} C_DIS
LIN {X 748.776, Y -447.822, Z 310.7, A 0, B 90, C -0, E1 0, E2 0, E3 0, E4 0} C_DIS
LIN {X 750.381, Y -449.09, Z 310.7, A 0, B 90, C -0, E1 0, E2 0, E3 0, E4 0} C_DIS
LIN {X 751.703, Y -450.688, Z 310.7, A 0, B 90, C -0, E1 0, E2 0, E3 0, E4 0} C_DIS
LIN {X 753.024, Y -452.287, Z 310.7, A 0, B 90, C -0, E1 0, E2 0, E3 0, E4 0} C_DIS
LIN {X 754.346, Y -453.885, Z 310.7, A 0, B 90, C -0, E1 0, E2 0, E3 0, E4 0} C_DIS
LIN {X 755.667, Y -455.484, Z 310.7, A 0, B 90, C -0, E1 0, E2 0, E3 0, E4 0} C_DIS
LIN {X 756.989, Y -457.082, Z 310.7, A 0, B 90, C -0, E1 0, E2 0, E3 0, E4 0} C_DIS
LIN {X 758.686, Y -458.119, Z 310.7, A 0, B 90, C -0, E1 0, E2 0, E3 0, E4 0} C_DIS
LIN {X 760.355, Y -456.977, Z 310.7, A 0, B 90, C -0, E1 0, E2 0, E3 0, E4 0} C_DIS
LIN {X 761.771, Y -455.461, Z 310.7, A 0, B 90, C -0, E1 0, E2 0, E3 0, E4 0} C_DIS
LIN {X 763.186, Y -453.945, Z 310.7, A 0, B 90, C -0, E1 0, E2 0, E3 0, E4 0} C_DIS
LIN {X 764.602, Y -452.429, Z 310.7, A 0, B 90, C -0, E1 0, E2 0, E3 0, E4 0} C_DIS
LIN {X 766.017, Y -450.913, Z 310.7, A 0, B 90, C -0, E1 0, E2 0, E3 0, E4 0} C_DIS
LIN {X 767.433, Y -449.397, Z 310.7, A 0, B 90, C -0, E1 0, E2 0, E3 0, E4 0} C_DIS
LIN {X 769.191, Y -448.366, Z 310.7, A 0, B 90, C -0, E1 0, E2 0, E3 0, E4 0} C_DIS
LIN {X 771.215, Y -448.662, Z 310.7, A 0, B 90, C -0, E1 0, E2 0, E3 0, E4 0} C_DIS
LIN {X 773.158, Y -449.386, Z 310.7, A 0, B 90, C -0, E1 0, E2 0, E3 0, E4 0} C_DIS
LIN {X 775.102, Y -450.109, Z 310.7, A 0, B 90, C -0, E1 0, E2 0, E3 0, E4 0} C_DIS
LIN {X 777.046, Y -450.833, Z 310.7, A 0, B 90, C -0, E1 0, E2 0, E3 0, E4 0} C_DIS
LIN {X 778.99, Y -451.556, Z 310.7, A 0, B 90, C -0, E1 0, E2 0, E3 0, E4 0} C_DIS
LIN {X 780.933, Y -452.28, Z 310.7, A 0, B 90, C -0, E1 0, E2 0, E3 0, E4 0} C_DIS
LIN {X 782.921, Y -452.329, Z 310.7, A 0, B 90, C -0, E1 0, E2 0, E3 0, E4 0} C_DIS
LIN {X 783.796, Y -450.506, Z 310.7, A 0, B 90, C -0, E1 0, E2 0, E3 0, E4 0} C_DIS
LIN {X 784.264, Y -448.485, Z 310.7, A 0, B 90, C -0, E1 0, E2 0, E3 0, E4 0} C_DIS
LIN {X 784.732, Y -446.465, Z 310.7, A 0, B 90, C -0, E1 0, E2 0, E3 0, E4 0} C_DIS
LIN {X 785.2, Y -444.444, Z 310.7, A 0, B 90, C -0, E1 0, E2 0, E3 0, E4 0} C_DIS
LIN {X 785.668, Y -442.423, Z 310.7, A 0, B 90, C -0, E1 0, E2 0, E3 0, E4 0} C_DIS
LIN {X 786.136, Y -440.403, Z 310.7, A 0, B 90, C -0, E1 0, E2 0, E3 0, E4 0} C_DIS
LIN {X 787.143, Y -438.631, Z 310.7, A 0, B 90, C -0, E1 0, E2 0, E3 0, E4 0} C_DIS
LIN {X 789.043, Y -437.875, Z 310.7, A 0, B 90, C -0, E1 0, E2 0, E3 0, E4 0} C_DIS
LIN {X 791.088, Y -437.53, Z 310.7, A 0, B 90, C -0, E1 0, E2 0, E3 0, E4 0} C_DIS
LIN {X 793.133, Y -437.185, Z 310.7, A 0, B 90, C -0, E1 0, E2 0, E3 0, E4 0} C_DIS
LIN {X 795.179, Y -436.839, Z 310.7, A 0, B 90, C -0, E1 0, E2 0, E3 0, E4 0} C_DIS
LIN {X 797.224, Y -436.494, Z 310.7, A 0, B 90, C -0, E1 0, E2 0, E3 0, E4 0} C_DIS
LIN {X 799.269, Y -436.149, Z 310.7, A 0, B 90, C -0, E1 0, E2 0, E3 0, E4 0} C_DIS
LIN {X 801.015, Y -435.198, Z 310.7, A 0, B 90, C -0, E1 0, E2 0, E3 0, E4 0} C_DIS
LIN {X 800.861, Y -433.181, Z 310.7, A 0, B 90, C -0, E1 0, E2 0, E3 0, E4 0} C_DIS
LIN {X 800.256, Y -431.197, Z 310.7, A 0, B 90, C -0, E1 0, E2 0, E3 0, E4 0} C_DIS
LIN {X 799.651, Y -429.213, Z 310.7, A 0, B 90, C -0, E1 0, E2 0, E3 0, E4 0} C_DIS
LIN {X 799.046, Y -427.229, Z 310.7, A 0, B 90, C -0, E1 0, E2 0, E3 0, E4 0} C_DIS
LIN {X 798.441, Y -425.245, Z 310.7, A 0, B 90, C -0, E1 0, E2 0, E3 0, E4 0} C_DIS
LIN {X 797.836, Y -423.262, Z 310.7, A 0, B 90, C -0, E1 0, E2 0, E3 0, E4 0} C_DIS
LIN {X 797.822, Y -421.224, Z 310.7, A 0, B 90, C -0, E1 0, E2 0, E3 0, E4 0} C_DIS
LIN {X 799.09, Y -419.619, Z 310.7, A 0, B 90, C -0, E1 0, E2 0, E3 0, E4 0} C_DIS
LIN {X 800.688, Y -418.297, Z 310.7, A 0, B 90, C -0, E1 0, E2 0, E3 0, E4 0} C_DIS
LIN {X 802.287, Y -416.976, Z 310.7, A 0, B 90, C -0, E1 0, E2 0, E3 0, E4 0} C_DIS
LIN {X 803.885, Y -415.654, Z 310.7, A 0, B 90, C -0, E1 0, E2 0, E3 0, E4 0} C_DIS
LIN {X 805.484, Y -414.333, Z 310.7, A 0, B 90, C -0, E1 0, E2 0, E3 0, E4 0} C_DIS
LIN {X 807.082, Y -413.011, Z 310.7, A 0, B 90, C -0, E1 0, E2 0, E3 0, E4 0} C_DIS
LIN {X 808.119, Y -411.314, Z 310.7, A 0, B 90, C -0, E1 0, E2 0, E3 0, E4 0} C_DIS
LIN {X 806.977, Y -409.645, Z 310.7, A 0, B 90, C -0, E1 0, E2 0, E3 0, E4 0} C_DIS
LIN {X 805.461, Y -408.229, Z 310.7, A 0, B 90, C -0, E1 0, E2 0, E3 0, E4 0} C_DIS
LIN {X 803.945, Y -406.814, Z 310.7, A 0, B 90, C -0, E1 0, E2 0, E3 0, E4 0} C_DIS
LIN {X 802.429, Y -405.398, Z 310.7, A 0, B 90, C -0, E1 0, E2 0, E3 0, E4 0} C_DIS
LIN {X 800.913, Y -403.983, Z 310.7, A 0, B 90, C -0, E1 0, E2 0, E3 0, E4 0} C_DIS
LIN {X 799.397, Y -402.567, Z 310.7, A 0, B 90, C -0, E1 0, E2 0, E3 0, E4 0} C_DIS
LIN {X 798.366, Y -400.809, Z 310.7, A 0, B 90, C -0, E1 0, E2 0, E3 0, E4 0} C_DIS
LIN {X 798.662, Y -398.785, Z 310.7, A 0, B 90, C -0, E1 0, E2 0, E3 0, E4 0} C_DIS
LIN {X 799.386, Y -396.842, Z 310.7, A 0, B 90, C -0, E1 0, E2 0, E3 0, E4 0} C_DIS
LIN {X 800.109, Y -394.898, Z 310.7, A 0, B 90, C -0, E1 0, E2 0, E3 0, E4 0} C_DIS
LIN {X 800.833, Y -392.954, Z 310.7, A 0, B 90, C -0, E1 0, E2 0, E3 0, E4 0} C_DIS
LIN {X 801.556, Y -391.01, Z 310.7, A 0, B 90, C -0, E1 0, E2 0, E3 0, E4 0} C_DIS
LIN {X 802.28, Y -389.067, Z 310.7, A 0, B 90, C -0, E1 0, E2 0, E3 0, E4 0} C_DIS
LIN {X 802.329, Y -387.079, Z 310.7, A 0, B 90, C -0, E1 0, E2 0, E3 0, E4 0} C_DIS
LIN {X 800.506, Y -386.204, Z 310.7, A 0, B 90, C -0, E1 0, E2 0, E3 0, E4 0} C_DIS
LIN {X 798.485, Y -385.736, Z 310.7, A 0, B 90, C -0, E1 0, E2 0, E3 0, E4 0} C_DIS
LIN {X 796.465, Y -385.268, Z 310.7, A 0, B 90, C -0, E1 0, E2 0, E3 0, E4 0} C_DIS
LIN {X 794.444, Y -384.8, Z 310.7, A 0, B 90, C -0, E1 0, E2 0, E3 0, E4 0} C_DIS
LIN {X 792.423, Y -384.332, Z 310.7, A 0, B 90, C -0, E1 0, E2 0, E3 0, E4 0} C_DIS
LIN {X 790.403, Y -383.864, Z 310.7, A 0, B 90, C -0, E1 0, E2 0, E3 0, E4 0} C_DIS
LIN {X 788.631, Y -382.857, Z 310.7, A 0, B 90, C -0, E1 0, E2 0, E3 0, E4 0} C_DIS
LIN {X 787.875, Y -380.957, Z 310.7, A 0, B 90, C -0, E1 0, E2 0, E3 0, E4 0} C_DIS
LIN {X 787.53, Y -378.912, Z 310.7, A 0, B 90, C -0, E1 0, E2 0, E3 0, E4 0} C_DIS
LIN {X 787.185, Y -376.867, Z 310.7, A 0, B 90, C -0, E1 0, E2 0, E3 0, E4 0} C_DIS
LIN {X 786.839, Y -374.821, Z 310.7, A 0, B 90, C -0, E1 0, E2 0, E3 0, E4 0} C_DIS
LIN {X 786.494, Y -372.776, Z 310.7, A 0, B 90, C -0, E1 0, E2 0, E3 0, E4 0} C_DIS
LIN {X 786.149, Y -370.731, Z 310.7, A 0, B 90, C -0, E1 0, E2 0, E3 0, E4 0} C_DIS
LIN {X 785.198, Y -368.985, Z 310.7, A 0, B 90, C -0, E1 0, E2 0, E3 0, E4 0} C_DIS
LIN {X 783.181, Y -369.139, Z 310.7, A 0, B 90, C -0, E1 0, E2 0, E3 0, E4 0} C_DIS
LIN {X 781.197, Y -369.744, Z 310.7, A 0, B 90, C -0, E1 0, E2 0, E3 0, E4 0} C_DIS
LIN {X 779.213, Y -370.349, Z 310.7, A 0, B 90, C -0, E1 0, E2 0, E3 0, E4 0} C_DIS
LIN {X 777.229, Y -370.954, Z 310.7, A 0, B 90, C -0, E1 0, E2 0, E3 0, E4 0} C_DIS
LIN {X 775.245, Y -371.559, Z 310.7, A 0, B 90, C -0, E1 0, E2 0, E3 0, E4 0} C_DIS
LIN {X 773.262, Y -372.164, Z 310.7, A 0, B 90, C -0, E1 0, E2 0, E3 0, E4 0} C_DIS
LIN {X 771.224, Y -372.178, Z 310.7, A 0, B 90, C -0, E1 0, E2 0, E3 0, E4 0} C_DIS
LIN {X 769.619, Y -370.91, Z 310.7, A 0, B 90, C -0, E1 0, E2 0, E3 0, E4 0} C_DIS
LIN {X 768.297, Y -369.312, Z 310.7, A 0, B 90, C -0, E1 0, E2 0, E3 0, E4 0} C_DIS
LIN {X 766.976, Y -367.713, Z 310.7, A 0, B 90, C -0, E1 0, E2 0, E3 0, E4 0} C_DIS
LIN {X 765.654, Y -366.115, Z 310.7, A 0, B 90, C -0, E1 0, E2 0, E3 0, E4 0} C_DIS
LIN {X 764.333, Y -364.516, Z 310.7, A 0, B 90, C -0, E1 0, E2 0, E3 0, E4 0} C_DIS
LIN {X 763.011, Y -362.918, Z 310.7, A 0, B 90, C -0, E1 0, E2 0, E3 0, E4 0} C_DIS
LIN {X 761.314, Y -361.881, Z 310.7, A 0, B 90, C -0, E1 0, E2 0, E3 0, E4 0} C_DIS
LIN {X 759.645, Y -363.023, Z 310.7, A 0, B 90, C -0, E1 0, E2 0, E3 0, E4 0} C_DIS
LIN {X 758.229, Y -364.539, Z 310.7, A 0, B 90, C -0, E1 0, E2 0, E3 0, E4 0} C_DIS
LIN {X 756.814, Y -366.055, Z 310.7, A 0, B 90, C -0, E1 0, E2 0, E3 0, E4 0} C_DIS
LIN {X 755.398, Y -367.571, Z 310.7, A 0, B 90, C -0, E1 0, E2 0, E3 0, E4 0} C_DIS
LIN {X 753.983, Y -369.087, Z 310.7, A 0, B 90, C -0, E1 0, E2 0, E3 0, E4 0} C_DIS
LIN {X 752.464, Y -370.615, Z 312, A 0, B 90, C -0, E1 0, E2 0, E3 0, E4 0} C_DIS
LIN {X 750.708, Y -371.651, Z 312, A 0, B 90, C -0, E1 0, E2 0, E3 0, E4 0} C_DIS
LIN {X 748.683, Y -371.36, Z 312, A 0, B 90, C -0, E1 0, E2 0, E3 0, E4 0} C_DIS
LIN {X 746.737, Y -370.642, Z 312, A 0, B 90, C -0, E1 0, E2 0, E3 0, E4 0} C_DIS
LIN {X 744.792, Y -369.923, Z 312, A 0, B 90, C -0, E1 0, E2 0, E3 0, E4 0} C_DIS
LIN {X 742.846, Y -369.204, Z 312, A 0, B 90, C -0, E1 0, E2 0, E3 0, E4 0} C_DIS
LIN {X 740.9, Y -368.486, Z 312, A 0, B 90, C -0, E1 0, E2 0, E3 0, E4 0} C_DIS
LIN {X 738.954, Y -367.767, Z 312, A 0, B 90, C -0, E1 0, E2 0, E3 0, E4 0} C_DIS
LIN {X 736.965, Y -367.723, Z 312, A 0, B 90, C -0, E1 0, E2 0, E3 0, E4 0} C_DIS
LIN {X 736.095, Y -369.549, Z 312, A 0, B 90, C -0, E1 0, E2 0, E3 0, E4 0} C_DIS
LIN {X 735.632, Y -371.571, Z 312, A 0, B 90, C -0, E1 0, E2 0, E3 0, E4 0} C_DIS
LIN {X 735.169, Y -373.593, Z 312, A 0, B 90, C -0, E1 0, E2 0, E3 0, E4 0} C_DIS
LIN {X 734.707, Y -375.616, Z 312, A 0, B 90, C -0, E1 0, E2 0, E3 0, E4 0} C_DIS
LIN {X 734.244, Y -377.638, Z 312, A 0, B 90, C -0, E1 0, E2 0, E3 0, E4 0} C_DIS
LIN {X 733.781, Y -379.66, Z 312, A 0, B 90, C -0, E1 0, E2 0, E3 0, E4 0} C_DIS
LIN {X 732.779, Y -381.435, Z 312, A 0, B 90, C -0, E1 0, E2 0, E3 0, E4 0} C_DIS
LIN {X 730.88, Y -382.195, Z 312, A 0, B 90, C -0, E1 0, E2 0, E3 0, E4 0} C_DIS
LIN {X 728.835, Y -382.546, Z 312, A 0, B 90, C -0, E1 0, E2 0, E3 0, E4 0} C_DIS
LIN {X 726.791, Y -382.897, Z 312, A 0, B 90, C -0, E1 0, E2 0, E3 0, E4 0} C_DIS
LIN {X 724.746, Y -383.247, Z 312, A 0, B 90, C -0, E1 0, E2 0, E3 0, E4 0} C_DIS
LIN {X 722.701, Y -383.598, Z 312, A 0, B 90, C -0, E1 0, E2 0, E3 0, E4 0} C_DIS
LIN {X 720.657, Y -383.948, Z 312, A 0, B 90, C -0, E1 0, E2 0, E3 0, E4 0} C_DIS
LIN {X 718.913, Y -384.904, Z 312, A 0, B 90, C -0, E1 0, E2 0, E3 0, E4 0} C_DIS
LIN {X 719.072, Y -386.921, Z 312, A 0, B 90, C -0, E1 0, E2 0, E3 0, E4 0} C_DIS
LIN {X 719.682, Y -388.904, Z 312, A 0, B 90, C -0, E1 0, E2 0, E3 0, E4 0} C_DIS
LIN {X 720.293, Y -390.886, Z 312, A 0, B 90, C -0, E1 0, E2 0, E3 0, E4 0} C_DIS
LIN {X 720.903, Y -392.869, Z 312, A 0, B 90, C -0, E1 0, E2 0, E3 0, E4 0} C_DIS
LIN {X 721.513, Y -394.852, Z 312, A 0, B 90, C -0, E1 0, E2 0, E3 0, E4 0} C_DIS
LIN {X 722.124, Y -396.834, Z 312, A 0, B 90, C -0, E1 0, E2 0, E3 0, E4 0} C_DIS
LIN {X 722.143, Y -398.872, Z 312, A 0, B 90, C -0, E1 0, E2 0, E3 0, E4 0} C_DIS
LIN {X 720.879, Y -400.481, Z 312, A 0, B 90, C -0, E1 0, E2 0, E3 0, E4 0} C_DIS
LIN {X 719.284, Y -401.807, Z 312, A 0, B 90, C -0, E1 0, E2 0, E3 0, E4 0} C_DIS
LIN {X 717.688, Y -403.133, Z 312, A 0, B 90, C -0, E1 0, E2 0, E3 0, E4 0} C_DIS
LIN {X 716.093, Y -404.458, Z 312, A 0, B 90, C -0, E1 0, E2 0, E3 0, E4 0} C_DIS
LIN {X 714.497, Y -405.784, Z 312, A 0, B 90, C -0, E1 0, E2 0, E3 0, E4 0} C_DIS
LIN {X 712.902, Y -407.11, Z 312, A 0, B 90, C -0, E1 0, E2 0, E3 0, E4 0} C_DIS
LIN {X 711.87, Y -408.81, Z 312, A 0, B 90, C -0, E1 0, E2 0, E3 0, E4 0} C_DIS
LIN {X 713.016, Y -410.477, Z 312, A 0, B 90, C -0, E1 0, E2 0, E3 0, E4 0} C_DIS
LIN {X 714.536, Y -411.889, Z 312, A 0, B 90, C -0, E1 0, E2 0, E3 0, E4 0} C_DIS
LIN {X 716.056, Y -413.301, Z 312, A 0, B 90, C -0, E1 0, E2 0, E3 0, E4 0} C_DIS
LIN {X 717.576, Y -414.713, Z 312, A 0, B 90, C -0, E1 0, E2 0, E3 0, E4 0} C_DIS
LIN {X 719.095, Y -416.124, Z 312, A 0, B 90, C -0, E1 0, E2 0, E3 0, E4 0} C_DIS
LIN {X 720.615, Y -417.536, Z 312, A 0, B 90, C -0, E1 0, E2 0, E3 0, E4 0} C_DIS
LIN {X 721.651, Y -419.292, Z 312, A 0, B 90, C -0, E1 0, E2 0, E3 0, E4 0} C_DIS
LIN {X 721.36, Y -421.316, Z 312, A 0, B 90, C -0, E1 0, E2 0, E3 0, E4 0} C_DIS
LIN {X 720.642, Y -423.262, Z 312, A 0, B 90, C -0, E1 0, E2 0, E3 0, E4 0} C_DIS
LIN {X 719.923, Y -425.208, Z 312, A 0, B 90, C -0, E1 0, E2 0, E3 0, E4 0} C_DIS
LIN {X 719.204, Y -427.154, Z 312, A 0, B 90, C -0, E1 0, E2 0, E3 0, E4 0} C_DIS
LIN {X 718.486, Y -429.1, Z 312, A 0, B 90, C -0, E1 0, E2 0, E3 0, E4 0} C_DIS
LIN {X 717.767, Y -431.046, Z 312, A 0, B 90, C -0, E1 0, E2 0, E3 0, E4 0} C_DIS
LIN {X 717.723, Y -433.035, Z 312, A 0, B 90, C -0, E1 0, E2 0, E3 0, E4 0} C_DIS
LIN {X 719.549, Y -433.905, Z 312, A 0, B 90, C -0, E1 0, E2 0, E3 0, E4 0} C_DIS
LIN {X 721.571, Y -434.368, Z 312, A 0, B 90, C -0, E1 0, E2 0, E3 0, E4 0} C_DIS
LIN {X 723.593, Y -434.831, Z 312, A 0, B 90, C -0, E1 0, E2 0, E3 0, E4 0} C_DIS
LIN {X 725.616, Y -435.293, Z 312, A 0, B 90, C -0, E1 0, E2 0, E3 0, E4 0} C_DIS
LIN {X 727.638, Y -435.756, Z 312, A 0, B 90, C -0, E1 0, E2 0, E3 0, E4 0} C_DIS
LIN {X 729.66, Y -436.219, Z 312, A 0, B 90, C -0, E1 0, E2 0, E3 0, E4 0} C_DIS
LIN {X 731.435, Y -437.221, Z 312, A 0, B 90, C -0, E1 0, E2 0, E3 0, E4 0} C_DIS
LIN {X 732.195, Y -439.12, Z 312, A 0, B 90, C -0, E1 0, E2 0, E3 0, E4 0} C_DIS
LIN {X 732.546, Y -441.165, Z 312, A 0, B 90, C -0, E1 0, E2 0, E3 0, E4 0} C_DIS
LIN {X 732.897, Y -443.209, Z 312, A 0, B 90, C -0, E1 0, E2 0, E3 0, E4 0} C_DIS
LIN {X 733.247, Y -445.254, Z 312, A 0, B 90, C -0, E1 0, E2 0, E3 0, E4 0} C_DIS
LIN {X 733.598, Y -447.299, Z 312, A 0, B 90, C -0, E1 0, E2 0, E3 0, E4 0} C_DIS
LIN {X 733.948, Y -449.343, Z 312, A 0, B 90, C -0, E1 0, E2 0, E3 0, E4 0} C_DIS
LIN {X 734.904, Y -451.087, Z 312, A 0, B 90, C -0, E1 0, E2 0, E3 0, E4 0} C_DIS
LIN {X 736.921, Y -450.928, Z 312, A 0, B 90, C -0, E1 0, E2 0, E3 0, E4 0} C_DIS
LIN {X 738.904, Y -450.318, Z 312, A 0, B 90, C -0, E1 0, E2 0, E3 0, E4 0} C_DIS
LIN {X 740.886, Y -449.707, Z 312, A 0, B 90, C -0, E1 0, E2 0, E3 0, E4 0} C_DIS
LIN {X 742.869, Y -449.097, Z 312, A 0, B 90, C -0, E1 0, E2 0, E3 0, E4 0} C_DIS
LIN {X 744.852, Y -448.487, Z 312, A 0, B 90, C -0, E1 0, E2 0, E3 0, E4 0} C_DIS
LIN {X 746.834, Y -447.876, Z 312, A 0, B 90, C -0, E1 0, E2 0, E3 0, E4 0} C_DIS
LIN {X 748.872, Y -447.857, Z 312, A 0, B 90, C -0, E1 0, E2 0, E3 0, E4 0} C_DIS
LIN {X 750.481, Y -449.121, Z 312, A 0, B 90, C -0, E1 0, E2 0, E3 0, E4 0} C_DIS
LIN {X 751.807, Y -450.716, Z 312, A 0, B 90, C -0, E1 0, E2 0, E3 0, E4 0} C_DIS
LIN {X 753.133, Y -452.312, Z 312, A 0, B 90, C -0, E1 0, E2 0, E3 0, E4 0} C_DIS
LIN {X 754.458, Y -453.907, Z 312, A 0, B 90, C -0, E1 0, E2 0, E3 0, E4 0} C_DIS
LIN {X 755.784, Y -455.503, Z 312, A 0, B 90, C -0, E1 0, E2 0, E3 0, E4 0} C_DIS
LIN {X 757.11, Y -457.098, Z 312, A 0, B 90, C -0, E1 0, E2 0, E3 0, E4 0} C_DIS
LIN {X 758.81, Y -458.13, Z 312, A 0, B 90, C -0, E1 0, E2 0, E3 0, E4 0} C_DIS
LIN {X 760.477, Y -456.984, Z 312, A 0, B 90, C -0, E1 0, E2 0, E3 0, E4 0} C_DIS
LIN {X 761.889, Y -455.464, Z 312, A 0, B 90, C -0, E1 0, E2 0, E3 0, E4 0} C_DIS
LIN {X 763.301, Y -453.944, Z 312, A 0, B 90, C -0, E1 0, E2 0, E3 0, E4 0} C_DIS
LIN {X 764.713, Y -452.424, Z 312, A 0, B 90, C -0, E1 0, E2 0, E3 0, E4 0} C_DIS
LIN {X 766.124, Y -450.905, Z 312, A 0, B 90, C -0, E1 0, E2 0, E3 0, E4 0} C_DIS
LIN {X 767.536, Y -449.385, Z 312, A 0, B 90, C -0, E1 0, E2 0, E3 0, E4 0} C_DIS
LIN {X 769.292, Y -448.349, Z 312, A 0, B 90, C -0, E1 0, E2 0, E3 0, E4 0} C_DIS
LIN {X 771.317, Y -448.64, Z 312, A 0, B 90, C -0, E1 0, E2 0, E3 0, E4 0} C_DIS
LIN {X 773.263, Y -449.358, Z 312, A 0, B 90, C -0, E1 0, E2 0, E3 0, E4 0} C_DIS
LIN {X 775.208, Y -450.077, Z 312, A 0, B 90, C -0, E1 0, E2 0, E3 0, E4 0} C_DIS
LIN {X 777.154, Y -450.796, Z 312, A 0, B 90, C -0, E1 0, E2 0, E3 0, E4 0} C_DIS
LIN {X 779.1, Y -451.514, Z 312, A 0, B 90, C -0, E1 0, E2 0, E3 0, E4 0} C_DIS
LIN {X 781.046, Y -452.233, Z 312, A 0, B 90, C -0, E1 0, E2 0, E3 0, E4 0} C_DIS
LIN {X 783.035, Y -452.277, Z 312, A 0, B 90, C -0, E1 0, E2 0, E3 0, E4 0} C_DIS
LIN {X 783.905, Y -450.451, Z 312, A 0, B 90, C -0, E1 0, E2 0, E3 0, E4 0} C_DIS
LIN {X 784.368, Y -448.429, Z 312, A 0, B 90, C -0, E1 0, E2 0, E3 0, E4 0} C_DIS
LIN {X 784.831, Y -446.407, Z 312, A 0, B 90, C -0, E1 0, E2 0, E3 0, E4 0} C_DIS
LIN {X 785.293, Y -444.384, Z 312, A 0, B 90, C -0, E1 0, E2 0, E3 0, E4 0} C_DIS
LIN {X 785.756, Y -442.362, Z 312, A 0, B 90, C -0, E1 0, E2 0, E3 0, E4 0} C_DIS
LIN {X 786.219, Y -440.34, Z 312, A 0, B 90, C -0, E1 0, E2 0, E3 0, E4 0} C_DIS
LIN {X 787.221, Y -438.565, Z 312, A 0, B 90, C -0, E1 0, E2 0, E3 0, E4 0} C_DIS
LIN {X 789.12, Y -437.805, Z 312, A 0, B 90, C -0, E1 0, E2 0, E3 0, E4 0} C_DIS
LIN {X 791.165, Y -437.454, Z 312, A 0, B 90, C -0, E1 0, E2 0, E3 0, E4 0} C_DIS
LIN {X 793.209, Y -437.103, Z 312, A 0, B 90, C -0, E1 0, E2 0, E3 0, E4 0} C_DIS
LIN {X 795.254, Y -436.753, Z 312, A 0, B 90, C -0, E1 0, E2 0, E3 0, E4 0} C_DIS
LIN {X 797.299, Y -436.402, Z 312, A 0, B 90, C -0, E1 0, E2 0, E3 0, E4 0} C_DIS
LIN {X 799.343, Y -436.052, Z 312, A 0, B 90, C -0, E1 0, E2 0, E3 0, E4 0} C_DIS
LIN {X 801.087, Y -435.096, Z 312, A 0, B 90, C -0, E1 0, E2 0, E3 0, E4 0} C_DIS
LIN {X 800.928, Y -433.079, Z 312, A 0, B 90, C -0, E1 0, E2 0, E3 0, E4 0} C_DIS
LIN {X 800.318, Y -431.096, Z 312, A 0, B 90, C -0, E1 0, E2 0, E3 0, E4 0} C_DIS
LIN {X 799.707, Y -429.114, Z 312, A 0, B 90, C -0, E1 0, E2 0, E3 0, E4 0} C_DIS
LIN {X 799.097, Y -427.131, Z 312, A 0, B 90, C -0, E1 0, E2 0, E3 0, E4 0} C_DIS
LIN {X 798.487, Y -425.148, Z 312, A 0, B 90, C -0, E1 0, E2 0, E3 0, E4 0} C_DIS
LIN {X 797.876, Y -423.166, Z 312, A 0, B 90, C -0, E1 0, E2 0, E3 0, E4 0} C_DIS
LIN {X 797.857, Y -421.128, Z 312, A 0, B 90, C -0, E1 0, E2 0, E3 0, E4 0} C_DIS
LIN {X 799.121, Y -419.519, Z 312, A 0, B 90, C -0, E1 0, E2 0, E3 0, E4 0} C_DIS
LIN {X 800.716, Y -418.193, Z 312, A 0, B 90, C -0, E1 0, E2 0, E3 0, E4 0} C_DIS
LIN {X 802.312, Y -416.867, Z 312, A 0, B 90, C -0, E1 0, E2 0, E3 0, E4 0} C_DIS
LIN {X 803.907, Y -415.542, Z 312, A 0, B 90, C -0, E1 0, E2 0, E3 0, E4 0} C_DIS
LIN {X 805.503, Y -414.216, Z 312, A 0, B 90, C -0, E1 0, E2 0, E3 0, E4 0} C_DIS
LIN {X 807.098, Y -412.89, Z 312, A 0, B 90, C -0, E1 0, E2 0, E3 0, E4 0} C_DIS
LIN {X 808.13, Y -411.19, Z 312, A 0, B 90, C -0, E1 0, E2 0, E3 0, E4 0} C_DIS
LIN {X 806.984, Y -409.523, Z 312, A 0, B 90, C -0, E1 0, E2 0, E3 0, E4 0} C_DIS
LIN {X 805.464, Y -408.111, Z 312, A 0, B 90, C -0, E1 0, E2 0, E3 0, E4 0} C_DIS
LIN {X 803.944, Y -406.699, Z 312, A 0, B 90, C -0, E1 0, E2 0, E3 0, E4 0} C_DIS
LIN {X 802.424, Y -405.287, Z 312, A 0, B 90, C -0, E1 0, E2 0, E3 0, E4 0} C_DIS
LIN {X 800.905, Y -403.876, Z 312, A 0, B 90, C -0, E1 0, E2 0, E3 0, E4 0} C_DIS
LIN {X 799.385, Y -402.464, Z 312, A 0, B 90, C -0, E1 0, E2 0, E3 0, E4 0} C_DIS
LIN {X 798.349, Y -400.708, Z 312, A 0, B 90, C -0, E1 0, E2 0, E3 0, E4 0} C_DIS
LIN {X 798.64, Y -398.684, Z 312, A 0, B 90, C -0, E1 0, E2 0, E3 0, E4 0} C_DIS
LIN {X 799.358, Y -396.738, Z 312, A 0, B 90, C -0, E1 0, E2 0, E3 0, E4 0} C_DIS
LIN {X 800.077, Y -394.792, Z 312, A 0, B 90, C -0, E1 0, E2 0, E3 0, E4 0} C_DIS
LIN {X 800.796, Y -392.846, Z 312, A 0, B 90, C -0, E1 0, E2 0, E3 0, E4 0} C_DIS
LIN {X 801.514, Y -390.9, Z 312, A 0, B 90, C -0, E1 0, E2 0, E3 0, E4 0} C_DIS
LIN {X 802.233, Y -388.954, Z 312, A 0, B 90, C -0, E1 0, E2 0, E3 0, E4 0} C_DIS
LIN {X 802.277, Y -386.965, Z 312, A 0, B 90, C -0, E1 0, E2 0, E3 0, E4 0} C_DIS
LIN {X 800.451, Y -386.095, Z 312, A 0, B 90, C -0, E1 0, E2 0, E3 0, E4 0} C_DIS
LIN {X 798.429, Y -385.632, Z 312, A 0, B 90, C -0, E1 0, E2 0, E3 0, E4 0} C_DIS
LIN {X 796.407, Y -385.169, Z 312, A 0, B 90, C -0, E1 0, E2 0, E3 0, E4 0} C_DIS
LIN {X 794.384, Y -384.707, Z 312, A 0, B 90, C -0, E1 0, E2 0, E3 0, E4 0} C_DIS
LIN {X 792.362, Y -384.244, Z 312, A 0, B 90, C -0, E1 0, E2 0, E3 0, E4 0} C_DIS
LIN {X 790.34, Y -383.781, Z 312, A 0, B 90, C -0, E1 0, E2 0, E3 0, E4 0} C_DIS
LIN {X 788.565, Y -382.779, Z 312, A 0, B 90, C -0, E1 0, E2 0, E3 0, E4 0} C_DIS
LIN {X 787.805, Y -380.88, Z 312, A 0, B 90, C -0, E1 0, E2 0, E3 0, E4 0} C_DIS
LIN {X 787.454, Y -378.835, Z 312, A 0, B 90, C -0, E1 0, E2 0, E3 0, E4 0} C_DIS
LIN {X 787.103, Y -376.791, Z 312, A 0, B 90, C -0, E1 0, E2 0, E3 0, E4 0} C_DIS
LIN {X 786.753, Y -374.746, Z 312, A 0, B 90, C -0, E1 0, E2 0, E3 0, E4 0} C_DIS
LIN {X 786.402, Y -372.701, Z 312, A 0, B 90, C -0, E1 0, E2 0, E3 0, E4 0} C_DIS
LIN {X 786.052, Y -370.657, Z 312, A 0, B 90, C -0, E1 0, E2 0, E3 0, E4 0} C_DIS
LIN {X 785.096, Y -368.913, Z 312, A 0, B 90, C -0, E1 0, E2 0, E3 0, E4 0} C_DIS
LIN {X 783.079, Y -369.072, Z 312, A 0, B 90, C -0, E1 0, E2 0, E3 0, E4 0} C_DIS
LIN {X 781.096, Y -369.682, Z 312, A 0, B 90, C -0, E1 0, E2 0, E3 0, E4 0} C_DIS
LIN {X 779.114, Y -370.293, Z 312, A 0, B 90, C -0, E1 0, E2 0, E3 0, E4 0} C_DIS
LIN {X 777.131, Y -370.903, Z 312, A 0, B 90, C -0, E1 0, E2 0, E3 0, E4 0} C_DIS
LIN {X 775.148, Y -371.513, Z 312, A 0, B 90, C -0, E1 0, E2 0, E3 0, E4 0} C_DIS
LIN {X 773.166, Y -372.124, Z 312, A 0, B 90, C -0, E1 0, E2 0, E3 0, E4 0} C_DIS
LIN {X 771.128, Y -372.143, Z 312, A 0, B 90, C -0, E1 0, E2 0, E3 0, E4 0} C_DIS
LIN {X 769.519, Y -370.879, Z 312, A 0, B 90, C -0, E1 0, E2 0, E3 0, E4 0} C_DIS
LIN {X 768.193, Y -369.284, Z 312, A 0, B 90, C -0, E1 0, E2 0, E3 0, E4 0} C_DIS
LIN {X 766.867, Y -367.688, Z 312, A 0, B 90, C -0, E1 0, E2 0, E3 0, E4 0} C_DIS
LIN {X 765.542, Y -366.093, Z 312, A 0, B 90, C -0, E1 0, E2 0, E3 0, E4 0} C_DIS
LIN {X 764.216, Y -364.497, Z 312, A 0, B 90, C -0, E1 0, E2 0, E3 0, E4 0} C_DIS
LIN {X 762.89, Y -362.902, Z 312, A 0, B 90, C -0, E1 0, E2 0, E3 0, E4 0} C_DIS
LIN {X 761.19, Y -361.87, Z 312, A 0, B 90, C -0, E1 0, E2 0, E3 0, E4 0} C_DIS
LIN {X 759.523, Y -363.016, Z 312, A 0, B 90, C -0, E1 0, E2 0, E3 0, E4 0} C_DIS
LIN {X 758.111, Y -364.536, Z 312, A 0, B 90, C -0, E1 0, E2 0, E3 0, E4 0} C_DIS
LIN {X 756.699, Y -366.056, Z 312, A 0, B 90, C -0, E1 0, E2 0, E3 0, E4 0} C_DIS
LIN {X 755.287, Y -367.576, Z 312, A 0, B 90, C -0, E1 0, E2 0, E3 0, E4 0} C_DIS
LIN {X 753.876, Y -369.095, Z 312, A 0, B 90, C -0, E1 0, E2 0, E3 0, E4 0} C_DIS
LIN {X 752.364, Y -370.624, Z 313.3, A 0, B 90, C -0, E1 0, E2 0, E3 0, E4 0} C_DIS
LIN {X 750.611, Y -371.665, Z 313.3, A 0, B 90, C -0, E1 0, E2 0, E3 0, E4 0} C_DIS
LIN {X 748.585, Y -371.379, Z 313.3, A 0, B 90, C -0, E1 0, E2 0, E3 0, E4 0} C_DIS
LIN {X 746.637, Y -370.665, Z 313.3, A 0, B 90, C -0, E1 0, E2 0, E3 0, E4 0} C_DIS
LIN {X 744.688, Y -369.951, Z 313.3, A 0, B 90, C -0, E1 0, E2 0, E3 0, E4 0} C_DIS
LIN {X 742.74, Y -369.237, Z 313.3, A 0, B 90, C -0, E1 0, E2 0, E3 0, E4 0} C_DIS
LIN {X 740.792, Y -368.523, Z 313.3, A 0, B 90, C -0, E1 0, E2 0, E3 0, E4 0} C_DIS
LIN {X 738.844, Y -367.809, Z 313.3, A 0, B 90, C -0, E1 0, E2 0, E3 0, E4 0} C_DIS
LIN {X 736.855, Y -367.77, Z 313.3, A 0, B 90, C -0, E1 0, E2 0, E3 0, E4 0} C_DIS
LIN {X 735.989, Y -369.599, Z 313.3, A 0, B 90, C -0, E1 0, E2 0, E3 0, E4 0} C_DIS
LIN {X 735.531, Y -371.622, Z 313.3, A 0, B 90, C -0, E1 0, E2 0, E3 0, E4 0} C_DIS
LIN {X 735.073, Y -373.646, Z 313.3, A 0, B 90, C -0, E1 0, E2 0, E3 0, E4 0} C_DIS
LIN {X 734.615, Y -375.67, Z 313.3, A 0, B 90, C -0, E1 0, E2 0, E3 0, E4 0} C_DIS
LIN {X 734.157, Y -377.694, Z 313.3, A 0, B 90, C -0, E1 0, E2 0, E3 0, E4 0} C_DIS
LIN {X 733.699, Y -379.718, Z 313.3, A 0, B 90, C -0, E1 0, E2 0, E3 0, E4 0} C_DIS
LIN {X 732.701, Y -381.495, Z 313.3, A 0, B 90, C -0, E1 0, E2 0, E3 0, E4 0} C_DIS
LIN {X 730.804, Y -382.261, Z 313.3, A 0, B 90, C -0, E1 0, E2 0, E3 0, E4 0} C_DIS
LIN {X 728.76, Y -382.617, Z 313.3, A 0, B 90, C -0, E1 0, E2 0, E3 0, E4 0} C_DIS
LIN {X 726.715, Y -382.972, Z 313.3, A 0, B 90, C -0, E1 0, E2 0, E3 0, E4 0} C_DIS
LIN {X 724.671, Y -383.328, Z 313.3, A 0, B 90, C -0, E1 0, E2 0, E3 0, E4 0} C_DIS
LIN {X 722.627, Y -383.684, Z 313.3, A 0, B 90, C -0, E1 0, E2 0, E3 0, E4 0} C_DIS
LIN {X 720.583, Y -384.04, Z 313.3, A 0, B 90, C -0, E1 0, E2 0, E3 0, E4 0} C_DIS
LIN {X 718.841, Y -385, Z 313.3, A 0, B 90, C -0, E1 0, E2 0, E3 0, E4 0} C_DIS
LIN {X 719.005, Y -387.017, Z 313.3, A 0, B 90, C -0, E1 0, E2 0, E3 0, E4 0} C_DIS
LIN {X 719.62, Y -388.999, Z 313.3, A 0, B 90, C -0, E1 0, E2 0, E3 0, E4 0} C_DIS
LIN {X 720.236, Y -390.98, Z 313.3, A 0, B 90, C -0, E1 0, E2 0, E3 0, E4 0} C_DIS
LIN {X 720.851, Y -392.962, Z 313.3, A 0, B 90, C -0, E1 0, E2 0, E3 0, E4 0} C_DIS
LIN {X 721.466, Y -394.943, Z 313.3, A 0, B 90, C -0, E1 0, E2 0, E3 0, E4 0} C_DIS
LIN {X 722.082, Y -396.925, Z 313.3, A 0, B 90, C -0, E1 0, E2 0, E3 0, E4 0} C_DIS
LIN {X 722.106, Y -398.964, Z 313.3, A 0, B 90, C -0, E1 0, E2 0, E3 0, E4 0} C_DIS
LIN {X 720.846, Y -400.575, Z 313.3, A 0, B 90, C -0, E1 0, E2 0, E3 0, E4 0} C_DIS
LIN {X 719.253, Y -401.906, Z 313.3, A 0, B 90, C -0, E1 0, E2 0, E3 0, E4 0} C_DIS
LIN {X 717.661, Y -403.236, Z 313.3, A 0, B 90, C -0, E1 0, E2 0, E3 0, E4 0} C_DIS
LIN {X 716.068, Y -404.566, Z 313.3, A 0, B 90, C -0, E1 0, E2 0, E3 0, E4 0} C_DIS
LIN {X 714.476, Y -405.896, Z 313.3, A 0, B 90, C -0, E1 0, E2 0, E3 0, E4 0} C_DIS
LIN {X 712.883, Y -407.226, Z 313.3, A 0, B 90, C -0, E1 0, E2 0, E3 0, E4 0} C_DIS
LIN {X 711.855, Y -408.929, Z 313.3, A 0, B 90, C -0, E1 0, E2 0, E3 0, E4 0} C_DIS
LIN {X 713.006, Y -410.594, Z 313.3, A 0, B 90, C -0, E1 0, E2 0, E3 0, E4 0} C_DIS
LIN {X 714.529, Y -412.002, Z 313.3, A 0, B 90, C -0, E1 0, E2 0, E3 0, E4 0} C_DIS
LIN {X 716.053, Y -413.41, Z 313.3, A 0, B 90, C -0, E1 0, E2 0, E3 0, E4 0} C_DIS
LIN {X 717.577, Y -414.819, Z 313.3, A 0, B 90, C -0, E1 0, E2 0, E3 0, E4 0} C_DIS
LIN {X 719.101, Y -416.227, Z 313.3, A 0, B 90, C -0, E1 0, E2 0, E3 0, E4 0} C_DIS
LIN {X 720.624, Y -417.636, Z 313.3, A 0, B 90, C -0, E1 0, E2 0, E3 0, E4 0} C_DIS
LIN {X 721.665, Y -419.389, Z 313.3, A 0, B 90, C -0, E1 0, E2 0, E3 0, E4 0} C_DIS
LIN {X 721.379, Y -421.415, Z 313.3, A 0, B 90, C -0, E1 0, E2 0, E3 0, E4 0} C_DIS
LIN {X 720.665, Y -423.363, Z 313.3, A 0, B 90, C -0, E1 0, E2 0, E3 0, E4 0} C_DIS
LIN {X 719.951, Y -425.312, Z 313.3, A 0, B 90, C -0, E1 0, E2 0, E3 0, E4 0} C_DIS
LIN {X 719.237, Y -427.26, Z 313.3, A 0, B 90, C -0, E1 0, E2 0, E3 0, E4 0} C_DIS
LIN {X 718.523, Y -429.208, Z 313.3, A 0, B 90, C -0, E1 0, E2 0, E3 0, E4 0} C_DIS
LIN {X 717.809, Y -431.156, Z 313.3, A 0, B 90, C -0, E1 0, E2 0, E3 0, E4 0} C_DIS
LIN {X 717.77, Y -433.145, Z 313.3, A 0, B 90, C -0, E1 0, E2 0, E3 0, E4 0} C_DIS
LIN {X 719.599, Y -434.011, Z 313.3, A 0, B 90, C -0, E1 0, E2 0, E3 0, E4 0} C_DIS
LIN {X 721.622, Y -434.469, Z 313.3, A 0, B 90, C -0, E1 0, E2 0, E3 0, E4 0} C_DIS
LIN {X 723.646, Y -434.927, Z 313.3, A 0, B 90, C -0, E1 0, E2 0, E3 0, E4 0} C_DIS
LIN {X 725.67, Y -435.385, Z 313.3, A 0, B 90, C -0, E1 0, E2 0, E3 0, E4 0} C_DIS
LIN {X 727.694, Y -435.843, Z 313.3, A 0, B 90, C -0, E1 0, E2 0, E3 0, E4 0} C_DIS
LIN {X 729.718, Y -436.301, Z 313.3, A 0, B 90, C -0, E1 0, E2 0, E3 0, E4 0} C_DIS
LIN {X 731.495, Y -437.299, Z 313.3, A 0, B 90, C -0, E1 0, E2 0, E3 0, E4 0} C_DIS
LIN {X 732.261, Y -439.196, Z 313.3, A 0, B 90, C -0, E1 0, E2 0, E3 0, E4 0} C_DIS
LIN {X 732.617, Y -441.24, Z 313.3, A 0, B 90, C -0, E1 0, E2 0, E3 0, E4 0} C_DIS
LIN {X 732.972, Y -443.285, Z 313.3, A 0, B 90, C -0, E1 0, E2 0, E3 0, E4 0} C_DIS
LIN {X 733.328, Y -445.329, Z 313.3, A 0, B 90, C -0, E1 0, E2 0, E3 0, E4 0} C_DIS
LIN {X 733.684, Y -447.373, Z 313.3, A 0, B 90, C -0, E1 0, E2 0, E3 0, E4 0} C_DIS
LIN {X 734.04, Y -449.417, Z 313.3, A 0, B 90, C -0, E1 0, E2 0, E3 0, E4 0} C_DIS
LIN {X 735, Y -451.159, Z 313.3, A 0, B 90, C -0, E1 0, E2 0, E3 0, E4 0} C_DIS
LIN {X 737.017, Y -450.995, Z 313.3, A 0, B 90, C -0, E1 0, E2 0, E3 0, E4 0} C_DIS
LIN {X 738.999, Y -450.38, Z 313.3, A 0, B 90, C -0, E1 0, E2 0, E3 0, E4 0} C_DIS
LIN {X 740.98, Y -449.764, Z 313.3, A 0, B 90, C -0, E1 0, E2 0, E3 0, E4 0} C_DIS
LIN {X 742.962, Y -449.149, Z 313.3, A 0, B 90, C -0, E1 0, E2 0, E3 0, E4 0} C_DIS
LIN {X 744.943, Y -448.534, Z 313.3, A 0, B 90, C -0, E1 0, E2 0, E3 0, E4 0} C_DIS
LIN {X 746.925, Y -447.918, Z 313.3, A 0, B 90, C -0, E1 0, E2 0, E3 0, E4 0} C_DIS
LIN {X 748.964, Y -447.894, Z 313.3, A 0, B 90, C -0, E1 0, E2 0, E3 0, E4 0} C_DIS
LIN {X 750.575, Y -449.154, Z 313.3, A 0, B 90, C -0, E1 0, E2 0, E3 0, E4 0} C_DIS
LIN {X 751.906, Y -450.747, Z 313.3, A 0, B 90, C -0, E1 0, E2 0, E3 0, E4 0} C_DIS
LIN {X 753.236, Y -452.339, Z 313.3, A 0, B 90, C -0, E1 0, E2 0, E3 0, E4 0} C_DIS
LIN {X 754.566, Y -453.932, Z 313.3, A 0, B 90, C -0, E1 0, E2 0, E3 0, E4 0} C_DIS
LIN {X 755.896, Y -455.524, Z 313.3, A 0, B 90, C -0, E1 0, E2 0, E3 0, E4 0} C_DIS
LIN {X 757.226, Y -457.117, Z 313.3, A 0, B 90, C -0, E1 0, E2 0, E3 0, E4 0} C_DIS
LIN {X 758.929, Y -458.145, Z 313.3, A 0, B 90, C -0, E1 0, E2 0, E3 0, E4 0} C_DIS
LIN {X 760.594, Y -456.994, Z 313.3, A 0, B 90, C -0, E1 0, E2 0, E3 0, E4 0} C_DIS
LIN {X 762.002, Y -455.471, Z 313.3, A 0, B 90, C -0, E1 0, E2 0, E3 0, E4 0} C_DIS
LIN {X 763.41, Y -453.947, Z 313.3, A 0, B 90, C -0, E1 0, E2 0, E3 0, E4 0} C_DIS
LIN {X 764.819, Y -452.423, Z 313.3, A 0, B 90, C -0, E1 0, E2 0, E3 0, E4 0} C_DIS
LIN {X 766.227, Y -450.899, Z 313.3, A 0, B 90, C -0, E1 0, E2 0, E3 0, E4 0} C_DIS
LIN {X 767.636, Y -449.376, Z 313.3, A 0, B 90, C -0, E1 0, E2 0, E3 0, E4 0} C_DIS
LIN {X 769.389, Y -448.335, Z 313.3, A 0, B 90, C -0, E1 0, E2 0, E3 0, E4 0} C_DIS
LIN {X 771.415, Y -448.621, Z 313.3, A 0, B 90, C -0, E1 0, E2 0, E3 0, E4 0} C_DIS
LIN {X 773.363, Y -449.335, Z 313.3, A 0, B 90, C -0, E1 0, E2 0, E3 0, E4 0} C_DIS
LIN {X 775.312, Y -450.049, Z 313.3, A 0, B 90, C -0, E1 0, E2 0, E3 0, E4 0} C_DIS
LIN {X 777.26, Y -450.763, Z 313.3, A 0, B 90, C -0, E1 0, E2 0, E3 0, E4 0} C_DIS
LIN {X 779.208, Y -451.477, Z 313.3, A 0, B 90, C -0, E1 0, E2 0, E3 0, E4 0} C_DIS
LIN {X 781.156, Y -452.191, Z 313.3, A 0, B 90, C -0, E1 0, E2 0, E3 0, E4 0} C_DIS
LIN {X 783.145, Y -452.23, Z 313.3, A 0, B 90, C -0, E1 0, E2 0, E3 0, E4 0} C_DIS
LIN {X 784.011, Y -450.401, Z 313.3, A 0, B 90, C -0, E1 0, E2 0, E3 0, E4 0} C_DIS
LIN {X 784.469, Y -448.378, Z 313.3, A 0, B 90, C -0, E1 0, E2 0, E3 0, E4 0} C_DIS
LIN {X 784.927, Y -446.354, Z 313.3, A 0, B 90, C -0, E1 0, E2 0, E3 0, E4 0} C_DIS
LIN {X 785.385, Y -444.33, Z 313.3, A 0, B 90, C -0, E1 0, E2 0, E3 0, E4 0} C_DIS
LIN {X 785.843, Y -442.306, Z 313.3, A 0, B 90, C -0, E1 0, E2 0, E3 0, E4 0} C_DIS
LIN {X 786.301, Y -440.282, Z 313.3, A 0, B 90, C -0, E1 0, E2 0, E3 0, E4 0} C_DIS
LIN {X 787.299, Y -438.505, Z 313.3, A 0, B 90, C -0, E1 0, E2 0, E3 0, E4 0} C_DIS
LIN {X 789.196, Y -437.739, Z 313.3, A 0, B 90, C -0, E1 0, E2 0, E3 0, E4 0} C_DIS
LIN {X 791.24, Y -437.383, Z 313.3, A 0, B 90, C -0, E1 0, E2 0, E3 0, E4 0} C_DIS
LIN {X 793.285, Y -437.028, Z 313.3, A 0, B 90, C -0, E1 0, E2 0, E3 0, E4 0} C_DIS
LIN {X 795.329, Y -436.672, Z 313.3, A 0, B 90, C -0, E1 0, E2 0, E3 0, E4 0} C_DIS
LIN {X 797.373, Y -436.316, Z 313.3, A 0, B 90, C -0, E1 0, E2 0, E3 0, E4 0} C_DIS
LIN {X 799.417, Y -435.96, Z 313.3, A 0, B 90, C -0, E1 0, E2 0, E3 0, E4 0} C_DIS
LIN {X 801.159, Y -435, Z 313.3, A 0, B 90, C -0, E1 0, E2 0, E3 0, E4 0} C_DIS
LIN {X 800.995, Y -432.983, Z 313.3, A 0, B 90, C -0, E1 0, E2 0, E3 0, E4 0} C_DIS
LIN {X 800.38, Y -431.001, Z 313.3, A 0, B 90, C -0, E1 0, E2 0, E3 0, E4 0} C_DIS
LIN {X 799.764, Y -429.02, Z 313.3, A 0, B 90, C -0, E1 0, E2 0, E3 0, E4 0} C_DIS
LIN {X 799.149, Y -427.038, Z 313.3, A 0, B 90, C -0, E1 0, E2 0, E3 0, E4 0} C_DIS
LIN {X 798.534, Y -425.057, Z 313.3, A 0, B 90, C -0, E1 0, E2 0, E3 0, E4 0} C_DIS
LIN {X 797.918, Y -423.075, Z 313.3, A 0, B 90, C -0, E1 0, E2 0, E3 0, E4 0} C_DIS
LIN {X 797.894, Y -421.036, Z 313.3, A 0, B 90, C -0, E1 0, E2 0, E3 0, E4 0} C_DIS
LIN {X 799.154, Y -419.425, Z 313.3, A 0, B 90, C -0, E1 0, E2 0, E3 0, E4 0} C_DIS
LIN {X 800.747, Y -418.094, Z 313.3, A 0, B 90, C -0, E1 0, E2 0, E3 0, E4 0} C_DIS
LIN {X 802.339, Y -416.764, Z 313.3, A 0, B 90, C -0, E1 0, E2 0, E3 0, E4 0} C_DIS
LIN {X 803.932, Y -415.434, Z 313.3, A 0, B 90, C -0, E1 0, E2 0, E3 0, E4 0} C_DIS
LIN {X 805.524, Y -414.104, Z 313.3, A 0, B 90, C -0, E1 0, E2 0, E3 0, E4 0} C_DIS
LIN {X 807.117, Y -412.774, Z 313.3, A 0, B 90, C -0, E1 0, E2 0, E3 0, E4 0} C_DIS
LIN {X 808.145, Y -411.071, Z 313.3, A 0, B 90, C -0, E1 0, E2 0, E3 0, E4 0} C_DIS
LIN {X 806.994, Y -409.406, Z 313.3, A 0, B 90, C -0, E1 0, E2 0, E3 0, E4 0} C_DIS
LIN {X 805.471, Y -407.998, Z 313.3, A 0, B 90, C -0, E1 0, E2 0, E3 0, E4 0} C_DIS
LIN {X 803.947, Y -406.59, Z 313.3, A 0, B 90, C -0, E1 0, E2 0, E3 0, E4 0} C_DIS
LIN {X 802.423, Y -405.181, Z 313.3, A 0, B 90, C -0, E1 0, E2 0, E3 0, E4 0} C_DIS
LIN {X 800.899, Y -403.773, Z 313.3, A 0, B 90, C -0, E1 0, E2 0, E3 0, E4 0} C_DIS
LIN {X 799.376, Y -402.364, Z 313.3, A 0, B 90, C -0, E1 0, E2 0, E3 0, E4 0} C_DIS
LIN {X 798.335, Y -400.611, Z 313.3, A 0, B 90, C -0, E1 0, E2 0, E3 0, E4 0} C_DIS
LIN {X 798.621, Y -398.585, Z 313.3, A 0, B 90, C -0, E1 0, E2 0, E3 0, E4 0} C_DIS
LIN {X 799.335, Y -396.637, Z 313.3, A 0, B 90, C -0, E1 0, E2 0, E3 0, E4 0} C_DIS
LIN {X 800.049, Y -394.688, Z 313.3, A 0, B 90, C -0, E1 0, E2 0, E3 0, E4 0} C_DIS
LIN {X 800.763, Y -392.74, Z 313.3, A 0, B 90, C -0, E1 0, E2 0, E3 0, E4 0} C_DIS
LIN {X 801.477, Y -390.792, Z 313.3, A 0, B 90, C -0, E1 0, E2 0, E3 0, E4 0} C_DIS
LIN {X 802.191, Y -388.844, Z 313.3, A 0, B 90, C -0, E1 0, E2 0, E3 0, E4 0} C_DIS
LIN {X 802.23, Y -386.855, Z 313.3, A 0, B 90, C -0, E1 0, E2 0, E3 0, E4 0} C_DIS
LIN {X 800.401, Y -385.989, Z 313.3, A 0, B 90, C -0, E1 0, E2 0, E3 0, E4 0} C_DIS
LIN {X 798.378, Y -385.531, Z 313.3, A 0, B 90, C -0, E1 0, E2 0, E3 0, E4 0} C_DIS
LIN {X 796.354, Y -385.073, Z 313.3, A 0, B 90, C -0, E1 0, E2 0, E3 0, E4 0} C_DIS
LIN {X 794.33, Y -384.615, Z 313.3, A 0, B 90, C -0, E1 0, E2 0, E3 0, E4 0} C_DIS
LIN {X 792.306, Y -384.157, Z 313.3, A 0, B 90, C -0, E1 0, E2 0, E3 0, E4 0} C_DIS
LIN {X 790.282, Y -383.699, Z 313.3, A 0, B 90, C -0, E1 0, E2 0, E3 0, E4 0} C_DIS
LIN {X 788.505, Y -382.701, Z 313.3, A 0, B 90, C -0, E1 0, E2 0, E3 0, E4 0} C_DIS
LIN {X 787.739, Y -380.804, Z 313.3, A 0, B 90, C -0, E1 0, E2 0, E3 0, E4 0} C_DIS
LIN {X 787.383, Y -378.76, Z 313.3, A 0, B 90, C -0, E1 0, E2 0, E3 0, E4 0} C_DIS
LIN {X 787.028, Y -376.715, Z 313.3, A 0, B 90, C -0, E1 0, E2 0, E3 0, E4 0} C_DIS
LIN {X 786.672, Y -374.671, Z 313.3, A 0, B 90, C -0, E1 0, E2 0, E3 0, E4 0} C_DIS
LIN {X 786.316, Y -372.627, Z 313.3, A 0, B 90, C -0, E1 0, E2 0, E3 0, E4 0} C_DIS
LIN {X 785.96, Y -370.583, Z 313.3, A 0, B 90, C -0, E1 0, E2 0, E3 0, E4 0} C_DIS
LIN {X 785, Y -368.841, Z 313.3, A 0, B 90, C -0, E1 0, E2 0, E3 0, E4 0} C_DIS
LIN {X 782.983, Y -369.005, Z 313.3, A 0, B 90, C -0, E1 0, E2 0, E3 0, E4 0} C_DIS
LIN {X 781.001, Y -369.62, Z 313.3, A 0, B 90, C -0, E1 0, E2 0, E3 0, E4 0} C_DIS
LIN {X 779.02, Y -370.236, Z 313.3, A 0, B 90, C -0, E1 0, E2 0, E3 0, E4 0} C_DIS
LIN {X 777.038, Y -370.851, Z 313.3, A 0, B 90, C -0, E1 0, E2 0, E3 0, E4 0} C_DIS
LIN {X 775.057, Y -371.466, Z 313.3, A 0, B 90, C -0, E1 0, E2 0, E3 0, E4 0} C_DIS
LIN {X 773.075, Y -372.082, Z 313.3, A 0, B 90, C -0, E1 0, E2 0, E3 0, E4 0} C_DIS
LIN {X 771.036, Y -372.106, Z 313.3, A 0, B 90, C -0, E1 0, E2 0, E3 0, E4 0} C_DIS
LIN {X 769.425, Y -370.846, Z 313.3, A 0, B 90, C -0, E1 0, E2 0, E3 0, E4 0} C_DIS
LIN {X 768.094, Y -369.253, Z 313.3, A 0, B 90, C -0, E1 0, E2 0, E3 0, E4 0} C_DIS
LIN {X 766.764, Y -367.661, Z 313.3, A 0, B 90, C -0, E1 0, E2 0, E3 0, E4 0} C_DIS
LIN {X 765.434, Y -366.068, Z 313.3, A 0, B 90, C -0, E1 0, E2 0, E3 0, E4 0} C_DIS
LIN {X 764.104, Y -364.476, Z 313.3, A 0, B 90, C -0, E1 0, E2 0, E3 0, E4 0} C_DIS
LIN {X 762.774, Y -362.883, Z 313.3, A 0, B 90, C -0, E1 0, E2 0, E3 0, E4 0} C_DIS
LIN {X 761.071, Y -361.855, Z 313.3, A 0, B 90, C -0, E1 0, E2 0, E3 0, E4 0} C_DIS
LIN {X 759.406, Y -363.006, Z 313.3, A 0, B 90, C -0, E1 0, E2 0, E3 0, E4 0} C_DIS
LIN {X 757.998, Y -364.529, Z 313.3, A 0, B 90, C -0, E1 0, E2 0, E3 0, E4 0} C_DIS
LIN {X 756.59, Y -366.053, Z 313.3, A 0, B 90, C -0, E1 0, E2 0, E3 0, E4 0} C_DIS
LIN {X 755.181, Y -367.577, Z 313.3, A 0, B 90, C -0, E1 0, E2 0, E3 0, E4 0} C_DIS
LIN {X 753.773, Y -369.101, Z 313.3, A 0, B 90, C -0, E1 0, E2 0, E3 0, E4 0} C_DIS
LIN {X 752.269, Y -370.63, Z 314.6, A 0, B 90, C -0, E1 0, E2 0, E3 0, E4 0} C_DIS
LIN {X 750.517, Y -371.675, Z 314.6, A 0, B 90, C -0, E1 0, E2 0, E3 0, E4 0} C_DIS
LIN {X 748.49, Y -371.394, Z 314.6, A 0, B 90, C -0, E1 0, E2 0, E3 0, E4 0} C_DIS
LIN {X 746.539, Y -370.684, Z 314.6, A 0, B 90, C -0, E1 0, E2 0, E3 0, E4 0} C_DIS
LIN {X 744.589, Y -369.975, Z 314.6, A 0, B 90, C -0, E1 0, E2 0, E3 0, E4 0} C_DIS
LIN {X 742.638, Y -369.265, Z 314.6, A 0, B 90, C -0, E1 0, E2 0, E3 0, E4 0} C_DIS
LIN {X 740.688, Y -368.555, Z 314.6, A 0, B 90, C -0, E1 0, E2 0, E3 0, E4 0} C_DIS
LIN {X 738.737, Y -367.846, Z 314.6, A 0, B 90, C -0, E1 0, E2 0, E3 0, E4 0} C_DIS
LIN {X 736.748, Y -367.811, Z 314.6, A 0, B 90, C -0, E1 0, E2 0, E3 0, E4 0} C_DIS
LIN {X 735.885, Y -369.643, Z 314.6, A 0, B 90, C -0, E1 0, E2 0, E3 0, E4 0} C_DIS
LIN {X 735.432, Y -371.668, Z 314.6, A 0, B 90, C -0, E1 0, E2 0, E3 0, E4 0} C_DIS
LIN {X 734.979, Y -373.694, Z 314.6, A 0, B 90, C -0, E1 0, E2 0, E3 0, E4 0} C_DIS
LIN {X 734.526, Y -375.719, Z 314.6, A 0, B 90, C -0, E1 0, E2 0, E3 0, E4 0} C_DIS
LIN {X 734.073, Y -377.745, Z 314.6, A 0, B 90, C -0, E1 0, E2 0, E3 0, E4 0} C_DIS
LIN {X 733.619, Y -379.77, Z 314.6, A 0, B 90, C -0, E1 0, E2 0, E3 0, E4 0} C_DIS
LIN {X 732.625, Y -381.551, Z 314.6, A 0, B 90, C -0, E1 0, E2 0, E3 0, E4 0} C_DIS
LIN {X 730.729, Y -382.321, Z 314.6, A 0, B 90, C -0, E1 0, E2 0, E3 0, E4 0} C_DIS
LIN {X 728.685, Y -382.682, Z 314.6, A 0, B 90, C -0, E1 0, E2 0, E3 0, E4 0} C_DIS
LIN {X 726.641, Y -383.043, Z 314.6, A 0, B 90, C -0, E1 0, E2 0, E3 0, E4 0} C_DIS
LIN {X 724.597, Y -383.403, Z 314.6, A 0, B 90, C -0, E1 0, E2 0, E3 0, E4 0} C_DIS
LIN {X 722.553, Y -383.764, Z 314.6, A 0, B 90, C -0, E1 0, E2 0, E3 0, E4 0} C_DIS
LIN {X 720.509, Y -384.125, Z 314.6, A 0, B 90, C -0, E1 0, E2 0, E3 0, E4 0} C_DIS
LIN {X 718.769, Y -385.09, Z 314.6, A 0, B 90, C -0, E1 0, E2 0, E3 0, E4 0} C_DIS
LIN {X 718.937, Y -387.107, Z 314.6, A 0, B 90, C -0, E1 0, E2 0, E3 0, E4 0} C_DIS
LIN {X 719.558, Y -389.088, Z 314.6, A 0, B 90, C -0, E1 0, E2 0, E3 0, E4 0} C_DIS
